    movel(p[x_c + 0.003071, y_c + 0.108854, z_c, rx, ry, rz], a, v)
    movel(p[x_c + 0.002863, y_c + 0.109126, z_c, rx, ry, rz], a, v)
    movel(p[x_c + 0.002653, y_c + 0.109393, z_c, rx, ry, rz], a, v)
    movel(p[x_c + 0.002442, y_c + 0.109655, z_c, rx, ry, rz], a, v)
    movel(p[x_c + 0.002230, y_c + 0.109912, z_c, rx, ry, rz], a, v)
    movel(p[x_c + 0.002017, y_c + 0.110165, z_c, rx, ry, rz], a, v)
    movel(p[x_c + 0.001803, y_c + 0.110413, z_c, rx, ry, rz], a, v)
    movel(p[x_c + 0.001589, y_c + 0.110656, z_c, rx, ry, rz], a, v)
    movel(p[x_c + 0.001373, y_c + 0.110893, z_c, rx, ry, rz], a, v)
    movel(p[x_c + 0.001157, y_c + 0.111126, z_c, rx, ry, rz], a, v)
    movel(p[x_c + 0.000939, y_c + 0.111354, z_c, rx, ry, rz], a, v)
    movel(p[x_c + 0.000722, y_c + 0.111576, z_c, rx, ry, rz], a, v)
    movel(p[x_c + 0.000503, y_c + 0.111793, z_c, rx, ry, rz], a, v)
    movel(p[x_c + 0.000284, y_c + 0.112005, z_c, rx, ry, rz], a, v)
    movel(p[x_c + 0.000064, y_c + 0.112211, z_c, rx, ry, rz], a, v)
    movel(p[x_c + -0.000156, y_c + 0.112412, z_c, rx, ry, rz], a, v)
    movel(p[x_c + -0.000377, y_c + 0.112608, z_c, rx, ry, rz], a, v)
    movel(p[x_c + -0.000598, y_c + 0.112798, z_c, rx, ry, rz], a, v)
    movel(p[x_c + -0.000820, y_c + 0.112982, z_c, rx, ry, rz], a, v)
    movel(p[x_c + -0.001042, y_c + 0.113161, z_c, rx, ry, rz], a, v)
    movel(p[x_c + -0.001264, y_c + 0.113334, z_c, rx, ry, rz], a, v)
    movel(p[x_c + -0.001487, y_c + 0.113501, z_c, rx, ry, rz], a, v)
    movel(p[x_c + -0.001709, y_c + 0.113662, z_c, rx, ry, rz], a, v)
    movel(p[x_c + -0.001932, y_c + 0.113818, z_c, rx, ry, rz], a, v)
    movel(p[x_c + -0.002155, y_c + 0.113967, z_c, rx, ry, rz], a, v)
    movel(p[x_c + -0.002378, y_c + 0.114111, z_c, rx, ry, rz], a, v)
    movel(p[x_c + -0.002600, y_c + 0.114248, z_c, rx, ry, rz], a, v)
    movel(p[x_c + -0.002823, y_c + 0.114380, z_c, rx, ry, rz], a, v)
    movel(p[x_c + -0.003046, y_c + 0.114505, z_c, rx, ry, rz], a, v)
    movel(p[x_c + -0.003268, y_c + 0.114624, z_c, rx, ry, rz], a, v)
    movel(p[x_c + -0.003491, y_c + 0.114737, z_c, rx, ry, rz], a, v)
    movel(p[x_c + -0.003491, y_c + 0.114737, z_c, rx, ry, rz], a, v)
    movel(p[x_c + -0.003766, y_c + 0.114868, z_c, rx, ry, rz], a, v)
    movel(p[x_c + -0.004040, y_c + 0.114986, z_c, rx, ry, rz], a, v)
    movel(p[x_c + -0.004311, y_c + 0.115094, z_c, rx, ry, rz], a, v)
    movel(p[x_c + -0.004579, y_c + 0.115189, z_c, rx, ry, rz], a, v)
    movel(p[x_c + -0.004844, y_c + 0.115274, z_c, rx, ry, rz], a, v)
    movel(p[x_c + -0.005105, y_c + 0.115347, z_c, rx, ry, rz], a, v)
    movel(p[x_c + -0.005364, y_c + 0.115408, z_c, rx, ry, rz], a, v)
    movel(p[x_c + -0.005619, y_c + 0.115459, z_c, rx, ry, rz], a, v)
    movel(p[x_c + -0.005870, y_c + 0.115499, z_c, rx, ry, rz], a, v)
    movel(p[x_c + -0.006117, y_c + 0.115529, z_c, rx, ry, rz], a, v)
    movel(p[x_c + -0.006360, y_c + 0.115547, z_c, rx, ry, rz], a, v)
    movel(p[x_c + -0.006599, y_c + 0.115556, z_c, rx, ry, rz], a, v)
    movel(p[x_c + -0.006833, y_c + 0.115553, z_c, rx, ry, rz], a, v)
    movel(p[x_c + -0.007062, y_c + 0.115541, z_c, rx, ry, rz], a, v)
    movel(p[x_c + -0.007287, y_c + 0.115519, z_c, rx, ry, rz], a, v)
    movel(p[x_c + -0.007506, y_c + 0.115486, z_c, rx, ry, rz], a, v)
    movel(p[x_c + -0.007720, y_c + 0.115444, z_c, rx, ry, rz], a, v)
    movel(p[x_c + -0.007929, y_c + 0.115393, z_c, rx, ry, rz], a, v)
    movel(p[x_c + -0.008132, y_c + 0.115331, z_c, rx, ry, rz], a, v)
    movel(p[x_c + -0.008329, y_c + 0.115261, z_c, rx, ry, rz], a, v)
    movel(p[x_c + -0.008521, y_c + 0.115181, z_c, rx, ry, rz], a, v)
    movel(p[x_c + -0.008705, y_c + 0.115092, z_c, rx, ry, rz], a, v)
    movel(p[x_c + -0.008884, y_c + 0.114994, z_c, rx, ry, rz], a, v)
    movel(p[x_c + -0.009056, y_c + 0.114887, z_c, rx, ry, rz], a, v)
    movel(p[x_c + -0.009221, y_c + 0.114771, z_c, rx, ry, rz], a, v)
    movel(p[x_c + -0.009379, y_c + 0.114647, z_c, rx, ry, rz], a, v)
    movel(p[x_c + -0.009530, y_c + 0.114514, z_c, rx, ry, rz], a, v)
    movel(p[x_c + -0.009674, y_c + 0.114373, z_c, rx, ry, rz], a, v)
    movel(p[x_c + -0.009809, y_c + 0.114224, z_c, rx, ry, rz], a, v)
    movel(p[x_c + -0.009938, y_c + 0.114066, z_c, rx, ry, rz], a, v)
    movel(p[x_c + -0.010058, y_c + 0.113901, z_c, rx, ry, rz], a, v)
    movel(p[x_c + -0.010170, y_c + 0.113728, z_c, rx, ry, rz], a, v)
    movel(p[x_c + -0.010274, y_c + 0.113547, z_c, rx, ry, rz], a, v)
    movel(p[x_c + -0.010369, y_c + 0.113359, z_c, rx, ry, rz], a, v)
    movel(p[x_c + -0.010456, y_c + 0.113164, z_c, rx, ry, rz], a, v)
    movel(p[x_c + -0.010533, y_c + 0.112961, z_c, rx, ry, rz], a, v)
    movel(p[x_c + -0.010602, y_c + 0.112751, z_c, rx, ry, rz], a, v)
    movel(p[x_c + -0.010661, y_c + 0.112534, z_c, rx, ry, rz], a, v)
    movel(p[x_c + -0.010711, y_c + 0.112310, z_c, rx, ry, rz], a, v)
    movel(p[x_c + -0.010751, y_c + 0.112079, z_c, rx, ry, rz], a, v)
    movel(p[x_c + -0.010782, y_c + 0.111842, z_c, rx, ry, rz], a, v)
    movel(p[x_c + -0.010802, y_c + 0.111598, z_c, rx, ry, rz], a, v)
    movel(p[x_c + -0.010812, y_c + 0.111349, z_c, rx, ry, rz], a, v)
    movel(p[x_c + -0.010812, y_c + 0.111092, z_c, rx, ry, rz], a, v)
    movel(p[x_c + -0.010801, y_c + 0.110830, z_c, rx, ry, rz], a, v)
    movel(p[x_c + -0.010779, y_c + 0.110562, z_c, rx, ry, rz], a, v)
    movel(p[x_c + -0.010746, y_c + 0.110288, z_c, rx, ry, rz], a, v)
    movel(p[x_c + -0.010702, y_c + 0.110008, z_c, rx, ry, rz], a, v)
    movel(p[x_c + -0.010647, y_c + 0.109723, z_c, rx, ry, rz], a, v)
    movel(p[x_c + -0.010647, y_c + 0.109723, z_c, rx, ry, rz], a, v)
    movel(p[x_c + -0.010635, y_c + 0.109670, z_c, rx, ry, rz], a, v)
    movel(p[x_c + -0.010621, y_c + 0.109614, z_c, rx, ry, rz], a, v)
    movel(p[x_c + -0.010606, y_c + 0.109555, z_c, rx, ry, rz], a, v)
    movel(p[x_c + -0.010588, y_c + 0.109492, z_c, rx, ry, rz], a, v)
    movel(p[x_c + -0.010569, y_c + 0.109426, z_c, rx, ry, rz], a, v)
    movel(p[x_c + -0.010548, y_c + 0.109356, z_c, rx, ry, rz], a, v)
    movel(p[x_c + -0.010525, y_c + 0.109284, z_c, rx, ry, rz], a, v)
    movel(p[x_c + -0.010501, y_c + 0.109209, z_c, rx, ry, rz], a, v)
    movel(p[x_c + -0.010475, y_c + 0.109130, z_c, rx, ry, rz], a, v)
    movel(p[x_c + -0.010447, y_c + 0.109049, z_c, rx, ry, rz], a, v)
    movel(p[x_c + -0.010417, y_c + 0.108965, z_c, rx, ry, rz], a, v)
    movel(p[x_c + -0.010386, y_c + 0.108878, z_c, rx, ry, rz], a, v)
    movel(p[x_c + -0.010353, y_c + 0.108788, z_c, rx, ry, rz], a, v)
    movel(p[x_c + -0.010318, y_c + 0.108695, z_c, rx, ry, rz], a, v)
    movel(p[x_c + -0.010282, y_c + 0.108600, z_c, rx, ry, rz], a, v)
    movel(p[x_c + -0.010244, y_c + 0.108502, z_c, rx, ry, rz], a, v)
    movel(p[x_c + -0.010205, y_c + 0.108401, z_c, rx, ry, rz], a, v)
    movel(p[x_c + -0.010164, y_c + 0.108298, z_c, rx, ry, rz], a, v)
    movel(p[x_c + -0.010122, y_c + 0.108192, z_c, rx, ry, rz], a, v)
    movel(p[x_c + -0.010078, y_c + 0.108084, z_c, rx, ry, rz], a, v)
    movel(p[x_c + -0.010033, y_c + 0.107973, z_c, rx, ry, rz], a, v)
    movel(p[x_c + -0.009986, y_c + 0.107860, z_c, rx, ry, rz], a, v)
    movel(p[x_c + -0.009938, y_c + 0.107745, z_c, rx, ry, rz], a, v)
    movel(p[x_c + -0.009888, y_c + 0.107627, z_c, rx, ry, rz], a, v)
    movel(p[x_c + -0.009837, y_c + 0.107507, z_c, rx, ry, rz], a, v)
    movel(p[x_c + -0.009784, y_c + 0.107385, z_c, rx, ry, rz], a, v)
    movel(p[x_c + -0.009731, y_c + 0.107261, z_c, rx, ry, rz], a, v)
    movel(p[x_c + -0.009676, y_c + 0.107135, z_c, rx, ry, rz], a, v)
    movel(p[x_c + -0.009619, y_c + 0.107007, z_c, rx, ry, rz], a, v)
    movel(p[x_c + -0.009561, y_c + 0.106877, z_c, rx, ry, rz], a, v)
    movel(p[x_c + -0.009503, y_c + 0.106744, z_c, rx, ry, rz], a, v)
    movel(p[x_c + -0.009442, y_c + 0.106610, z_c, rx, ry, rz], a, v)
    movel(p[x_c + -0.009381, y_c + 0.106475, z_c, rx, ry, rz], a, v)
    movel(p[x_c + -0.009318, y_c + 0.106337, z_c, rx, ry, rz], a, v)
    movel(p[x_c + -0.009254, y_c + 0.106198, z_c, rx, ry, rz], a, v)
    movel(p[x_c + -0.009189, y_c + 0.106057, z_c, rx, ry, rz], a, v)
    movel(p[x_c + -0.009123, y_c + 0.105914, z_c, rx, ry, rz], a, v)
    movel(p[x_c + -0.009056, y_c + 0.105770, z_c, rx, ry, rz], a, v)
    movel(p[x_c + -0.008988, y_c + 0.105624, z_c, rx, ry, rz], a, v)
    movel(p[x_c + -0.008918, y_c + 0.105476, z_c, rx, ry, rz], a, v)
    movel(p[x_c + -0.008848, y_c + 0.105328, z_c, rx, ry, rz], a, v)
    movel(p[x_c + -0.008776, y_c + 0.105178, z_c, rx, ry, rz], a, v)
    movel(p[x_c + -0.008704, y_c + 0.105026, z_c, rx, ry, rz], a, v)
    movel(p[x_c + -0.008630, y_c + 0.104873, z_c, rx, ry, rz], a, v)
    movel(p[x_c + -0.008555, y_c + 0.104719, z_c, rx, ry, rz], a, v)
    movel(p[x_c + -0.008480, y_c + 0.104564, z_c, rx, ry, rz], a, v)
    movel(p[x_c + -0.008403, y_c + 0.104408, z_c, rx, ry, rz], a, v)
    movel(p[x_c + -0.008326, y_c + 0.104251, z_c, rx, ry, rz], a, v)
    movel(p[x_c + -0.008248, y_c + 0.104092, z_c, rx, ry, rz], a, v)
    movel(p[x_c + -0.008248, y_c + 0.104092, z_c, rx, ry, rz], a, v)
    movel(p[x_c + -0.008098, y_c + 0.103789, z_c, rx, ry, rz], a, v)
    movel(p[x_c + -0.007954, y_c + 0.103496, z_c, rx, ry, rz], a, v)
    movel(p[x_c + -0.007814, y_c + 0.103212, z_c, rx, ry, rz], a, v)
    movel(p[x_c + -0.007679, y_c + 0.102937, z_c, rx, ry, rz], a, v)
    movel(p[x_c + -0.007549, y_c + 0.102670, z_c, rx, ry, rz], a, v)
    movel(p[x_c + -0.007424, y_c + 0.102412, z_c, rx, ry, rz], a, v)
    movel(p[x_c + -0.007303, y_c + 0.102162, z_c, rx, ry, rz], a, v)
    movel(p[x_c + -0.007187, y_c + 0.101920, z_c, rx, ry, rz], a, v)
    movel(p[x_c + -0.007075, y_c + 0.101686, z_c, rx, ry, rz], a, v)
    movel(p[x_c + -0.006968, y_c + 0.101459, z_c, rx, ry, rz], a, v)
    movel(p[x_c + -0.006864, y_c + 0.101239, z_c, rx, ry, rz], a, v)
    movel(p[x_c + -0.006765, y_c + 0.101026, z_c, rx, ry, rz], a, v)
    movel(p[x_c + -0.006670, y_c + 0.100820, z_c, rx, ry, rz], a, v)
    movel(p[x_c + -0.006578, y_c + 0.100620, z_c, rx, ry, rz], a, v)
    movel(p[x_c + -0.006491, y_c + 0.100427, z_c, rx, ry, rz], a, v)
    movel(p[x_c + -0.006407, y_c + 0.100240, z_c, rx, ry, rz], a, v)
    movel(p[x_c + -0.006327, y_c + 0.100058, z_c, rx, ry, rz], a, v)
    movel(p[x_c + -0.006251, y_c + 0.099882, z_c, rx, ry, rz], a, v)
    movel(p[x_c + -0.006178, y_c + 0.099711, z_c, rx, ry, rz], a, v)
    movel(p[x_c + -0.006108, y_c + 0.099545, z_c, rx, ry, rz], a, v)
    movel(p[x_c + -0.006042, y_c + 0.099384, z_c, rx, ry, rz], a, v)
    movel(p[x_c + -0.005979, y_c + 0.099227, z_c, rx, ry, rz], a, v)
    movel(p[x_c + -0.005919, y_c + 0.099075, z_c, rx, ry, rz], a, v)
    movel(p[x_c + -0.005862, y_c + 0.098926, z_c, rx, ry, rz], a, v)
    movel(p[x_c + -0.005808, y_c + 0.098782, z_c, rx, ry, rz], a, v)
    movel(p[x_c + -0.005756, y_c + 0.098641, z_c, rx, ry, rz], a, v)
    movel(p[x_c + -0.005708, y_c + 0.098503, z_c, rx, ry, rz], a, v)
    movel(p[x_c + -0.005662, y_c + 0.098368, z_c, rx, ry, rz], a, v)
    movel(p[x_c + -0.005619, y_c + 0.098236, z_c, rx, ry, rz], a, v)
    movel(p[x_c + -0.005578, y_c + 0.098107, z_c, rx, ry, rz], a, v)
    movel(p[x_c + -0.005540, y_c + 0.097980, z_c, rx, ry, rz], a, v)
    movel(p[x_c + -0.005504, y_c + 0.097855, z_c, rx, ry, rz], a, v)
    movel(p[x_c + -0.005470, y_c + 0.097732, z_c, rx, ry, rz], a, v)
    movel(p[x_c + -0.005438, y_c + 0.097610, z_c, rx, ry, rz], a, v)
    movel(p[x_c + -0.005408, y_c + 0.097490, z_c, rx, ry, rz], a, v)
    movel(p[x_c + -0.005381, y_c + 0.097371, z_c, rx, ry, rz], a, v)
    movel(p[x_c + -0.005355, y_c + 0.097253, z_c, rx, ry, rz], a, v)
    movel(p[x_c + -0.005331, y_c + 0.097136, z_c, rx, ry, rz], a, v)
    movel(p[x_c + -0.005308, y_c + 0.097018, z_c, rx, ry, rz], a, v)
    movel(p[x_c + -0.005287, y_c + 0.096901, z_c, rx, ry, rz], a, v)
    movel(p[x_c + -0.005268, y_c + 0.096784, z_c, rx, ry, rz], a, v)
    movel(p[x_c + -0.005250, y_c + 0.096667, z_c, rx, ry, rz], a, v)
    movel(p[x_c + -0.005233, y_c + 0.096549, z_c, rx, ry, rz], a, v)
    movel(p[x_c + -0.005217, y_c + 0.096430, z_c, rx, ry, rz], a, v)
    movel(p[x_c + -0.005203, y_c + 0.096310, z_c, rx, ry, rz], a, v)
    movel(p[x_c + -0.005189, y_c + 0.096188, z_c, rx, ry, rz], a, v)
    movel(p[x_c + -0.005177, y_c + 0.096065, z_c, rx, ry, rz], a, v)
    movel(p[x_c + -0.005165, y_c + 0.095941, z_c, rx, ry, rz], a, v)
    movel(p[x_c + -0.005154, y_c + 0.095814, z_c, rx, ry, rz], a, v)
    movel(p[x_c + -0.005154, y_c + 0.095814, z_c, rx, ry, rz], a, v)
    movel(p[x_c + -0.005139, y_c + 0.095611, z_c, rx, ry, rz], a, v)
    movel(p[x_c + -0.005127, y_c + 0.095410, z_c, rx, ry, rz], a, v)
    movel(p[x_c + -0.005119, y_c + 0.095210, z_c, rx, ry, rz], a, v)
    movel(p[x_c + -0.005114, y_c + 0.095010, z_c, rx, ry, rz], a, v)
    movel(p[x_c + -0.005113, y_c + 0.094812, z_c, rx, ry, rz], a, v)
    movel(p[x_c + -0.005115, y_c + 0.094615, z_c, rx, ry, rz], a, v)
    movel(p[x_c + -0.005120, y_c + 0.094419, z_c, rx, ry, rz], a, v)
    movel(p[x_c + -0.005129, y_c + 0.094224, z_c, rx, ry, rz], a, v)
    movel(p[x_c + -0.005141, y_c + 0.094030, z_c, rx, ry, rz], a, v)
    movel(p[x_c + -0.005156, y_c + 0.093837, z_c, rx, ry, rz], a, v)
    movel(p[x_c + -0.005175, y_c + 0.093646, z_c, rx, ry, rz], a, v)
    movel(p[x_c + -0.005197, y_c + 0.093455, z_c, rx, ry, rz], a, v)
    movel(p[x_c + -0.005223, y_c + 0.093266, z_c, rx, ry, rz], a, v)
    movel(p[x_c + -0.005252, y_c + 0.093077, z_c, rx, ry, rz], a, v)
    movel(p[x_c + -0.005284, y_c + 0.092890, z_c, rx, ry, rz], a, v)
    movel(p[x_c + -0.005320, y_c + 0.092704, z_c, rx, ry, rz], a, v)
    movel(p[x_c + -0.005359, y_c + 0.092519, z_c, rx, ry, rz], a, v)
    movel(p[x_c + -0.005401, y_c + 0.092335, z_c, rx, ry, rz], a, v)
    movel(p[x_c + -0.005447, y_c + 0.092153, z_c, rx, ry, rz], a, v)
    movel(p[x_c + -0.005496, y_c + 0.091971, z_c, rx, ry, rz], a, v)
    movel(p[x_c + -0.005548, y_c + 0.091791, z_c, rx, ry, rz], a, v)
    movel(p[x_c + -0.005604, y_c + 0.091612, z_c, rx, ry, rz], a, v)
    movel(p[x_c + -0.005663, y_c + 0.091434, z_c, rx, ry, rz], a, v)
    movel(p[x_c + -0.005726, y_c + 0.091257, z_c, rx, ry, rz], a, v)
    movel(p[x_c + -0.005792, y_c + 0.091082, z_c, rx, ry, rz], a, v)
    movel(p[x_c + -0.005861, y_c + 0.090907, z_c, rx, ry, rz], a, v)
    movel(p[x_c + -0.005934, y_c + 0.090734, z_c, rx, ry, rz], a, v)
    movel(p[x_c + -0.006010, y_c + 0.090562, z_c, rx, ry, rz], a, v)
    movel(p[x_c + -0.006089, y_c + 0.090392, z_c, rx, ry, rz], a, v)
    movel(p[x_c + -0.006171, y_c + 0.090222, z_c, rx, ry, rz], a, v)
    movel(p[x_c + -0.006257, y_c + 0.090054, z_c, rx, ry, rz], a, v)
    movel(p[x_c + -0.006347, y_c + 0.089887, z_c, rx, ry, rz], a, v)
    movel(p[x_c + -0.006439, y_c + 0.089721, z_c, rx, ry, rz], a, v)
    movel(p[x_c + -0.006535, y_c + 0.089556, z_c, rx, ry, rz], a, v)
    movel(p[x_c + -0.006634, y_c + 0.089393, z_c, rx, ry, rz], a, v)
    movel(p[x_c + -0.006737, y_c + 0.089231, z_c, rx, ry, rz], a, v)
    movel(p[x_c + -0.006843, y_c + 0.089070, z_c, rx, ry, rz], a, v)
    movel(p[x_c + -0.006952, y_c + 0.088911, z_c, rx, ry, rz], a, v)
    movel(p[x_c + -0.007064, y_c + 0.088752, z_c, rx, ry, rz], a, v)
    movel(p[x_c + -0.007180, y_c + 0.088595, z_c, rx, ry, rz], a, v)
    movel(p[x_c + -0.007299, y_c + 0.088440, z_c, rx, ry, rz], a, v)
    movel(p[x_c + -0.007422, y_c + 0.088285, z_c, rx, ry, rz], a, v)
    movel(p[x_c + -0.007547, y_c + 0.088132, z_c, rx, ry, rz], a, v)
    movel(p[x_c + -0.007677, y_c + 0.087980, z_c, rx, ry, rz], a, v)
    movel(p[x_c + -0.007809, y_c + 0.087830, z_c, rx, ry, rz], a, v)
    movel(p[x_c + -0.007945, y_c + 0.087681, z_c, rx, ry, rz], a, v)
    movel(p[x_c + -0.008083, y_c + 0.087533, z_c, rx, ry, rz], a, v)
    movel(p[x_c + -0.008226, y_c + 0.087386, z_c, rx, ry, rz], a, v)
    movel(p[x_c + -0.008371, y_c + 0.087241, z_c, rx, ry, rz], a, v)
    movel(p[x_c + -0.008371, y_c + 0.087241, z_c, rx, ry, rz], a, v)
    movel(p[x_c + -0.008488, y_c + 0.087127, z_c, rx, ry, rz], a, v)
    movel(p[x_c + -0.008605, y_c + 0.087016, z_c, rx, ry, rz], a, v)
    movel(p[x_c + -0.008723, y_c + 0.086906, z_c, rx, ry, rz], a, v)
    movel(p[x_c + -0.008842, y_c + 0.086798, z_c, rx, ry, rz], a, v)
    movel(p[x_c + -0.008961, y_c + 0.086692, z_c, rx, ry, rz], a, v)
    movel(p[x_c + -0.009082, y_c + 0.086587, z_c, rx, ry, rz], a, v)
    movel(p[x_c + -0.009203, y_c + 0.086484, z_c, rx, ry, rz], a, v)
    movel(p[x_c + -0.009326, y_c + 0.086383, z_c, rx, ry, rz], a, v)
    movel(p[x_c + -0.009450, y_c + 0.086283, z_c, rx, ry, rz], a, v)
    movel(p[x_c + -0.009576, y_c + 0.086184, z_c, rx, ry, rz], a, v)
    movel(p[x_c + -0.009704, y_c + 0.086087, z_c, rx, ry, rz], a, v)
    movel(p[x_c + -0.009833, y_c + 0.085990, z_c, rx, ry, rz], a, v)
    movel(p[x_c + -0.009964, y_c + 0.085895, z_c, rx, ry, rz], a, v)
    movel(p[x_c + -0.010098, y_c + 0.085801, z_c, rx, ry, rz], a, v)
    movel(p[x_c + -0.010233, y_c + 0.085708, z_c, rx, ry, rz], a, v)
    movel(p[x_c + -0.010371, y_c + 0.085616, z_c, rx, ry, rz], a, v)
    movel(p[x_c + -0.010512, y_c + 0.085525, z_c, rx, ry, rz], a, v)
    movel(p[x_c + -0.010655, y_c + 0.085435, z_c, rx, ry, rz], a, v)
    movel(p[x_c + -0.010800, y_c + 0.085345, z_c, rx, ry, rz], a, v)
    movel(p[x_c + -0.010949, y_c + 0.085256, z_c, rx, ry, rz], a, v)
    movel(p[x_c + -0.011101, y_c + 0.085168, z_c, rx, ry, rz], a, v)
    movel(p[x_c + -0.011256, y_c + 0.085080, z_c, rx, ry, rz], a, v)
    movel(p[x_c + -0.011414, y_c + 0.084993, z_c, rx, ry, rz], a, v)
    movel(p[x_c + -0.011575, y_c + 0.084905, z_c, rx, ry, rz], a, v)
    movel(p[x_c + -0.011740, y_c + 0.084819, z_c, rx, ry, rz], a, v)
    movel(p[x_c + -0.011909, y_c + 0.084732, z_c, rx, ry, rz], a, v)
    movel(p[x_c + -0.012082, y_c + 0.084646, z_c, rx, ry, rz], a, v)
    movel(p[x_c + -0.012258, y_c + 0.084560, z_c, rx, ry, rz], a, v)
    movel(p[x_c + -0.012439, y_c + 0.084473, z_c, rx, ry, rz], a, v)
    movel(p[x_c + -0.012624, y_c + 0.084387, z_c, rx, ry, rz], a, v)
    movel(p[x_c + -0.012813, y_c + 0.084301, z_c, rx, ry, rz], a, v)
    movel(p[x_c + -0.013007, y_c + 0.084214, z_c, rx, ry, rz], a, v)
    movel(p[x_c + -0.013205, y_c + 0.084127, z_c, rx, ry, rz], a, v)
    movel(p[x_c + -0.013408, y_c + 0.084040, z_c, rx, ry, rz], a, v)
    movel(p[x_c + -0.013616, y_c + 0.083953, z_c, rx, ry, rz], a, v)
    movel(p[x_c + -0.013829, y_c + 0.083865, z_c, rx, ry, rz], a, v)
    movel(p[x_c + -0.014047, y_c + 0.083776, z_c, rx, ry, rz], a, v)
    movel(p[x_c + -0.014270, y_c + 0.083687, z_c, rx, ry, rz], a, v)
    movel(p[x_c + -0.014499, y_c + 0.083597, z_c, rx, ry, rz], a, v)
    movel(p[x_c + -0.014733, y_c + 0.083507, z_c, rx, ry, rz], a, v)
    movel(p[x_c + -0.014973, y_c + 0.083416, z_c, rx, ry, rz], a, v)
    movel(p[x_c + -0.015219, y_c + 0.083323, z_c, rx, ry, rz], a, v)
    movel(p[x_c + -0.015471, y_c + 0.083230, z_c, rx, ry, rz], a, v)
    movel(p[x_c + -0.015729, y_c + 0.083136, z_c, rx, ry, rz], a, v)
    movel(p[x_c + -0.015993, y_c + 0.083041, z_c, rx, ry, rz], a, v)
    movel(p[x_c + -0.016263, y_c + 0.082944, z_c, rx, ry, rz], a, v)
    movel(p[x_c + -0.016540, y_c + 0.082846, z_c, rx, ry, rz], a, v)
    movel(p[x_c + -0.016824, y_c + 0.082747, z_c, rx, ry, rz], a, v)
    movel(p[x_c + -0.017114, y_c + 0.082647, z_c, rx, ry, rz], a, v)
    movel(p[x_c + -0.017114, y_c + 0.082647, z_c, rx, ry, rz], a, v)
    movel(p[x_c + -0.017237, y_c + 0.082604, z_c, rx, ry, rz], a, v)
    movel(p[x_c + -0.017361, y_c + 0.082562, z_c, rx, ry, rz], a, v)
    movel(p[x_c + -0.017484, y_c + 0.082519, z_c, rx, ry, rz], a, v)
    movel(p[x_c + -0.017607, y_c + 0.082476, z_c, rx, ry, rz], a, v)
    movel(p[x_c + -0.017729, y_c + 0.082433, z_c, rx, ry, rz], a, v)
    movel(p[x_c + -0.017852, y_c + 0.082390, z_c, rx, ry, rz], a, v)
    movel(p[x_c + -0.017973, y_c + 0.082347, z_c, rx, ry, rz], a, v)
    movel(p[x_c + -0.018094, y_c + 0.082305, z_c, rx, ry, rz], a, v)
    movel(p[x_c + -0.018215, y_c + 0.082262, z_c, rx, ry, rz], a, v)
    movel(p[x_c + -0.018335, y_c + 0.082219, z_c, rx, ry, rz], a, v)
    movel(p[x_c + -0.018454, y_c + 0.082177, z_c, rx, ry, rz], a, v)
    movel(p[x_c + -0.018572, y_c + 0.082134, z_c, rx, ry, rz], a, v)
    movel(p[x_c + -0.018689, y_c + 0.082092, z_c, rx, ry, rz], a, v)
    movel(p[x_c + -0.018805, y_c + 0.082051, z_c, rx, ry, rz], a, v)
    movel(p[x_c + -0.018919, y_c + 0.082009, z_c, rx, ry, rz], a, v)
    movel(p[x_c + -0.019033, y_c + 0.081968, z_c, rx, ry, rz], a, v)
    movel(p[x_c + -0.019145, y_c + 0.081927, z_c, rx, ry, rz], a, v)
    movel(p[x_c + -0.019256, y_c + 0.081886, z_c, rx, ry, rz], a, v)
    movel(p[x_c + -0.019366, y_c + 0.081846, z_c, rx, ry, rz], a, v)
    movel(p[x_c + -0.019474, y_c + 0.081806, z_c, rx, ry, rz], a, v)
    movel(p[x_c + -0.019580, y_c + 0.081767, z_c, rx, ry, rz], a, v)
    movel(p[x_c + -0.019685, y_c + 0.081728, z_c, rx, ry, rz], a, v)
    movel(p[x_c + -0.019788, y_c + 0.081690, z_c, rx, ry, rz], a, v)
    movel(p[x_c + -0.019889, y_c + 0.081652, z_c, rx, ry, rz], a, v)
    movel(p[x_c + -0.019988, y_c + 0.081615, z_c, rx, ry, rz], a, v)
    movel(p[x_c + -0.020085, y_c + 0.081578, z_c, rx, ry, rz], a, v)
    movel(p[x_c + -0.020180, y_c + 0.081542, z_c, rx, ry, rz], a, v)
    movel(p[x_c + -0.020273, y_c + 0.081506, z_c, rx, ry, rz], a, v)
    movel(p[x_c + -0.020363, y_c + 0.081472, z_c, rx, ry, rz], a, v)
    movel(p[x_c + -0.020451, y_c + 0.081438, z_c, rx, ry, rz], a, v)
    movel(p[x_c + -0.020537, y_c + 0.081405, z_c, rx, ry, rz], a, v)
    movel(p[x_c + -0.020620, y_c + 0.081372, z_c, rx, ry, rz], a, v)
    movel(p[x_c + -0.020701, y_c + 0.081340, z_c, rx, ry, rz], a, v)
    movel(p[x_c + -0.020779, y_c + 0.081310, z_c, rx, ry, rz], a, v)
    movel(p[x_c + -0.020855, y_c + 0.081280, z_c, rx, ry, rz], a, v)
    movel(p[x_c + -0.020927, y_c + 0.081251, z_c, rx, ry, rz], a, v)
    movel(p[x_c + -0.020997, y_c + 0.081223, z_c, rx, ry, rz], a, v)
    movel(p[x_c + -0.021064, y_c + 0.081195, z_c, rx, ry, rz], a, v)
    movel(p[x_c + -0.021127, y_c + 0.081169, z_c, rx, ry, rz], a, v)
    movel(p[x_c + -0.021188, y_c + 0.081144, z_c, rx, ry, rz], a, v)
    movel(p[x_c + -0.021245, y_c + 0.081120, z_c, rx, ry, rz], a, v)
    movel(p[x_c + -0.021299, y_c + 0.081097, z_c, rx, ry, rz], a, v)
    movel(p[x_c + -0.021350, y_c + 0.081075, z_c, rx, ry, rz], a, v)
    movel(p[x_c + -0.021397, y_c + 0.081054, z_c, rx, ry, rz], a, v)
    movel(p[x_c + -0.021441, y_c + 0.081034, z_c, rx, ry, rz], a, v)
    movel(p[x_c + -0.021481, y_c + 0.081016, z_c, rx, ry, rz], a, v)
    movel(p[x_c + -0.021517, y_c + 0.080999, z_c, rx, ry, rz], a, v)
    movel(p[x_c + -0.021550, y_c + 0.080983, z_c, rx, ry, rz], a, v)
    movel(p[x_c + -0.021579, y_c + 0.080968, z_c, rx, ry, rz], a, v)
    movel(p[x_c + -0.021579, y_c + 0.080968, z_c, rx, ry, rz], a, v)
    movel(p[x_c + -0.022375, y_c + 0.080552, z_c, rx, ry, rz], a, v)
    movel(p[x_c + -0.022375, y_c + 0.080552, z_c, rx, ry, rz], a, v)
    movel(p[x_c + -0.020813, y_c + 0.080676, z_c, rx, ry, rz], a, v)
    movel(p[x_c + -0.020813, y_c + 0.080676, z_c, rx, ry, rz], a, v)
    movel(p[x_c + -0.020726, y_c + 0.080682, z_c, rx, ry, rz], a, v)
    movel(p[x_c + -0.020631, y_c + 0.080688, z_c, rx, ry, rz], a, v)
    movel(p[x_c + -0.020530, y_c + 0.080692, z_c, rx, ry, rz], a, v)
    movel(p[x_c + -0.020422, y_c + 0.080697, z_c, rx, ry, rz], a, v)
    movel(p[x_c + -0.020307, y_c + 0.080700, z_c, rx, ry, rz], a, v)
    movel(p[x_c + -0.020184, y_c + 0.080703, z_c, rx, ry, rz], a, v)
    movel(p[x_c + -0.020055, y_c + 0.080704, z_c, rx, ry, rz], a, v)
    movel(p[x_c + -0.019919, y_c + 0.080706, z_c, rx, ry, rz], a, v)
    movel(p[x_c + -0.019775, y_c + 0.080706, z_c, rx, ry, rz], a, v)
    movel(p[x_c + -0.019625, y_c + 0.080706, z_c, rx, ry, rz], a, v)
    movel(p[x_c + -0.019466, y_c + 0.080705, z_c, rx, ry, rz], a, v)
    movel(p[x_c + -0.019301, y_c + 0.080703, z_c, rx, ry, rz], a, v)
    movel(p[x_c + -0.019128, y_c + 0.080700, z_c, rx, ry, rz], a, v)
    movel(p[x_c + -0.018948, y_c + 0.080697, z_c, rx, ry, rz], a, v)
    movel(p[x_c + -0.018760, y_c + 0.080692, z_c, rx, ry, rz], a, v)
    movel(p[x_c + -0.018565, y_c + 0.080688, z_c, rx, ry, rz], a, v)
    movel(p[x_c + -0.018362, y_c + 0.080682, z_c, rx, ry, rz], a, v)
    movel(p[x_c + -0.018152, y_c + 0.080675, z_c, rx, ry, rz], a, v)
    movel(p[x_c + -0.017933, y_c + 0.080668, z_c, rx, ry, rz], a, v)
    movel(p[x_c + -0.017707, y_c + 0.080660, z_c, rx, ry, rz], a, v)
    movel(p[x_c + -0.017474, y_c + 0.080651, z_c, rx, ry, rz], a, v)
    movel(p[x_c + -0.017232, y_c + 0.080642, z_c, rx, ry, rz], a, v)
    movel(p[x_c + -0.016982, y_c + 0.080632, z_c, rx, ry, rz], a, v)
    movel(p[x_c + -0.016724, y_c + 0.080620, z_c, rx, ry, rz], a, v)
    movel(p[x_c + -0.016459, y_c + 0.080609, z_c, rx, ry, rz], a, v)
    movel(p[x_c + -0.016185, y_c + 0.080596, z_c, rx, ry, rz], a, v)
    movel(p[x_c + -0.015903, y_c + 0.080582, z_c, rx, ry, rz], a, v)
    movel(p[x_c + -0.015613, y_c + 0.080568, z_c, rx, ry, rz], a, v)
    movel(p[x_c + -0.015314, y_c + 0.080553, z_c, rx, ry, rz], a, v)
    movel(p[x_c + -0.015008, y_c + 0.080537, z_c, rx, ry, rz], a, v)
    movel(p[x_c + -0.014693, y_c + 0.080520, z_c, rx, ry, rz], a, v)
    movel(p[x_c + -0.014369, y_c + 0.080503, z_c, rx, ry, rz], a, v)
    movel(p[x_c + -0.014037, y_c + 0.080485, z_c, rx, ry, rz], a, v)
    movel(p[x_c + -0.013697, y_c + 0.080466, z_c, rx, ry, rz], a, v)
    movel(p[x_c + -0.013348, y_c + 0.080446, z_c, rx, ry, rz], a, v)
    movel(p[x_c + -0.012990, y_c + 0.080425, z_c, rx, ry, rz], a, v)
    movel(p[x_c + -0.012624, y_c + 0.080403, z_c, rx, ry, rz], a, v)
    movel(p[x_c + -0.012249, y_c + 0.080381, z_c, rx, ry, rz], a, v)
    movel(p[x_c + -0.011865, y_c + 0.080358, z_c, rx, ry, rz], a, v)
    movel(p[x_c + -0.011472, y_c + 0.080334, z_c, rx, ry, rz], a, v)
    movel(p[x_c + -0.011070, y_c + 0.080309, z_c, rx, ry, rz], a, v)
    movel(p[x_c + -0.010660, y_c + 0.080283, z_c, rx, ry, rz], a, v)
    movel(p[x_c + -0.010240, y_c + 0.080257, z_c, rx, ry, rz], a, v)
    movel(p[x_c + -0.009811, y_c + 0.080230, z_c, rx, ry, rz], a, v)
    movel(p[x_c + -0.009374, y_c + 0.080201, z_c, rx, ry, rz], a, v)
    movel(p[x_c + -0.008927, y_c + 0.080172, z_c, rx, ry, rz], a, v)
    movel(p[x_c + -0.008471, y_c + 0.080143, z_c, rx, ry, rz], a, v)
    movel(p[x_c + -0.008005, y_c + 0.080112, z_c, rx, ry, rz], a, v)
    movel(p[x_c + -0.007530, y_c + 0.080080, z_c, rx, ry, rz], a, v)
    movel(p[x_c + -0.007530, y_c + 0.080080, z_c, rx, ry, rz], a, v)
    movel(p[x_c + -0.007298, y_c + 0.080065, z_c, rx, ry, rz], a, v)
    movel(p[x_c + -0.007064, y_c + 0.080051, z_c, rx, ry, rz], a, v)
    movel(p[x_c + -0.006828, y_c + 0.080037, z_c, rx, ry, rz], a, v)
    movel(p[x_c + -0.006591, y_c + 0.080024, z_c, rx, ry, rz], a, v)
    movel(p[x_c + -0.006353, y_c + 0.080011, z_c, rx, ry, rz], a, v)
    movel(p[x_c + -0.006115, y_c + 0.079999, z_c, rx, ry, rz], a, v)
    movel(p[x_c + -0.005875, y_c + 0.079988, z_c, rx, ry, rz], a, v)
    movel(p[x_c + -0.005635, y_c + 0.079977, z_c, rx, ry, rz], a, v)
    movel(p[x_c + -0.005395, y_c + 0.079967, z_c, rx, ry, rz], a, v)
    movel(p[x_c + -0.005155, y_c + 0.079958, z_c, rx, ry, rz], a, v)
    movel(p[x_c + -0.004915, y_c + 0.079949, z_c, rx, ry, rz], a, v)
    movel(p[x_c + -0.004675, y_c + 0.079941, z_c, rx, ry, rz], a, v)
    movel(p[x_c + -0.004436, y_c + 0.079934, z_c, rx, ry, rz], a, v)
    movel(p[x_c + -0.004198, y_c + 0.079927, z_c, rx, ry, rz], a, v)
    movel(p[x_c + -0.003960, y_c + 0.079921, z_c, rx, ry, rz], a, v)
    movel(p[x_c + -0.003724, y_c + 0.079916, z_c, rx, ry, rz], a, v)
    movel(p[x_c + -0.003489, y_c + 0.079911, z_c, rx, ry, rz], a, v)
    movel(p[x_c + -0.003255, y_c + 0.079907, z_c, rx, ry, rz], a, v)
    movel(p[x_c + -0.003023, y_c + 0.079903, z_c, rx, ry, rz], a, v)
    movel(p[x_c + -0.002793, y_c + 0.079900, z_c, rx, ry, rz], a, v)
    movel(p[x_c + -0.002565, y_c + 0.079898, z_c, rx, ry, rz], a, v)
    movel(p[x_c + -0.002339, y_c + 0.079896, z_c, rx, ry, rz], a, v)
    movel(p[x_c + -0.002116, y_c + 0.079895, z_c, rx, ry, rz], a, v)
    movel(p[x_c + -0.001895, y_c + 0.079895, z_c, rx, ry, rz], a, v)
    movel(p[x_c + -0.001678, y_c + 0.079895, z_c, rx, ry, rz], a, v)
    movel(p[x_c + -0.001463, y_c + 0.079896, z_c, rx, ry, rz], a, v)
    movel(p[x_c + -0.001252, y_c + 0.079898, z_c, rx, ry, rz], a, v)
    movel(p[x_c + -0.001044, y_c + 0.079900, z_c, rx, ry, rz], a, v)
    movel(p[x_c + -0.000840, y_c + 0.079903, z_c, rx, ry, rz], a, v)
    movel(p[x_c + -0.000640, y_c + 0.079906, z_c, rx, ry, rz], a, v)
    movel(p[x_c + -0.000443, y_c + 0.079910, z_c, rx, ry, rz], a, v)
    movel(p[x_c + -0.000251, y_c + 0.079915, z_c, rx, ry, rz], a, v)
    movel(p[x_c + -0.000064, y_c + 0.079920, z_c, rx, ry, rz], a, v)
    movel(p[x_c + 0.000119, y_c + 0.079926, z_c, rx, ry, rz], a, v)
    movel(p[x_c + 0.000297, y_c + 0.079933, z_c, rx, ry, rz], a, v)
    movel(p[x_c + 0.000470, y_c + 0.079940, z_c, rx, ry, rz], a, v)
    movel(p[x_c + 0.000638, y_c + 0.079948, z_c, rx, ry, rz], a, v)
    movel(p[x_c + 0.000800, y_c + 0.079957, z_c, rx, ry, rz], a, v)
    movel(p[x_c + 0.000957, y_c + 0.079966, z_c, rx, ry, rz], a, v)
    movel(p[x_c + 0.001108, y_c + 0.079976, z_c, rx, ry, rz], a, v)
    movel(p[x_c + 0.001253, y_c + 0.079986, z_c, rx, ry, rz], a, v)
    movel(p[x_c + 0.001392, y_c + 0.079998, z_c, rx, ry, rz], a, v)
    movel(p[x_c + 0.001524, y_c + 0.080009, z_c, rx, ry, rz], a, v)
    movel(p[x_c + 0.001650, y_c + 0.080022, z_c, rx, ry, rz], a, v)
    movel(p[x_c + 0.001769, y_c + 0.080035, z_c, rx, ry, rz], a, v)
    movel(p[x_c + 0.001881, y_c + 0.080048, z_c, rx, ry, rz], a, v)
    movel(p[x_c + 0.001985, y_c + 0.080063, z_c, rx, ry, rz], a, v)
    movel(p[x_c + 0.002083, y_c + 0.080077, z_c, rx, ry, rz], a, v)
    movel(p[x_c + 0.002172, y_c + 0.080093, z_c, rx, ry, rz], a, v)
    movel(p[x_c + 0.002172, y_c + 0.080093, z_c, rx, ry, rz], a, v)
    movel(p[x_c + 0.002172, y_c + 0.080093, z_c, rx, ry, rz], a, v)
    movel(p[x_c + 0.002172, y_c + 0.080093, z_c, rx, ry, rz], a, v)
    movel(p[x_c + 0.002172, y_c + 0.080093, z_c, rx, ry, rz], a, v)
    movel(p[x_c + 0.002172, y_c + 0.080093, z_c, rx, ry, rz], a, v)
    movel(p[x_c + 0.002172, y_c + 0.080093, z_c, rx, ry, rz], a, v)
    movel(p[x_c + 0.002172, y_c + 0.080093, z_c, rx, ry, rz], a, v)
    movel(p[x_c + 0.002172, y_c + 0.080093, z_c, rx, ry, rz], a, v)
    movel(p[x_c + 0.002172, y_c + 0.080094, z_c, rx, ry, rz], a, v)
    movel(p[x_c + 0.002172, y_c + 0.080094, z_c, rx, ry, rz], a, v)
    movel(p[x_c + -0.072957, y_c + 0.089770, z_c, rx, ry, rz], a, v)
    movel(p[x_c + -0.072957, y_c + 0.089770, z_c, rx, ry, rz], a, v)
    movel(p[x_c + -0.072957, y_c + 0.089770, z_c, rx, ry, rz], a, v)
    movel(p[x_c + -0.072957, y_c + 0.089770, z_c, rx, ry, rz], a, v)
    movel(p[x_c + -0.072957, y_c + 0.089770, z_c, rx, ry, rz], a, v)
    movel(p[x_c + -0.072957, y_c + 0.089770, z_c, rx, ry, rz], a, v)
    movel(p[x_c + -0.072957, y_c + 0.089770, z_c, rx, ry, rz], a, v)
    movel(p[x_c + -0.072957, y_c + 0.089770, z_c, rx, ry, rz], a, v)
    movel(p[x_c + -0.072957, y_c + 0.089770, z_c, rx, ry, rz], a, v)
    movel(p[x_c + -0.072957, y_c + 0.089770, z_c, rx, ry, rz], a, v)
    movel(p[x_c + -0.072957, y_c + 0.089770, z_c, rx, ry, rz], a, v)
    movel(p[x_c + -0.072450, y_c + 0.089935, z_c, rx, ry, rz], a, v)
    movel(p[x_c + -0.071947, y_c + 0.090098, z_c, rx, ry, rz], a, v)
    movel(p[x_c + -0.071450, y_c + 0.090258, z_c, rx, ry, rz], a, v)
    movel(p[x_c + -0.070956, y_c + 0.090416, z_c, rx, ry, rz], a, v)
    movel(p[x_c + -0.070468, y_c + 0.090571, z_c, rx, ry, rz], a, v)
    movel(p[x_c + -0.069984, y_c + 0.090724, z_c, rx, ry, rz], a, v)
    movel(p[x_c + -0.069504, y_c + 0.090874, z_c, rx, ry, rz], a, v)
    movel(p[x_c + -0.069030, y_c + 0.091021, z_c, rx, ry, rz], a, v)
    movel(p[x_c + -0.068559, y_c + 0.091166, z_c, rx, ry, rz], a, v)
    movel(p[x_c + -0.068094, y_c + 0.091308, z_c, rx, ry, rz], a, v)
    movel(p[x_c + -0.067633, y_c + 0.091448, z_c, rx, ry, rz], a, v)
    movel(p[x_c + -0.067176, y_c + 0.091586, z_c, rx, ry, rz], a, v)
    movel(p[x_c + -0.066724, y_c + 0.091720, z_c, rx, ry, rz], a, v)
    movel(p[x_c + -0.066277, y_c + 0.091853, z_c, rx, ry, rz], a, v)
    movel(p[x_c + -0.065833, y_c + 0.091982, z_c, rx, ry, rz], a, v)
    movel(p[x_c + -0.065395, y_c + 0.092110, z_c, rx, ry, rz], a, v)
    movel(p[x_c + -0.064961, y_c + 0.092234, z_c, rx, ry, rz], a, v)
    movel(p[x_c + -0.064531, y_c + 0.092356, z_c, rx, ry, rz], a, v)
    movel(p[x_c + -0.064105, y_c + 0.092476, z_c, rx, ry, rz], a, v)
    movel(p[x_c + -0.063684, y_c + 0.092593, z_c, rx, ry, rz], a, v)
    movel(p[x_c + -0.063268, y_c + 0.092708, z_c, rx, ry, rz], a, v)
    movel(p[x_c + -0.062855, y_c + 0.092820, z_c, rx, ry, rz], a, v)
    movel(p[x_c + -0.062447, y_c + 0.092930, z_c, rx, ry, rz], a, v)
    movel(p[x_c + -0.062044, y_c + 0.093037, z_c, rx, ry, rz], a, v)
    movel(p[x_c + -0.061644, y_c + 0.093142, z_c, rx, ry, rz], a, v)
    movel(p[x_c + -0.061249, y_c + 0.093244, z_c, rx, ry, rz], a, v)
    movel(p[x_c + -0.060858, y_c + 0.093344, z_c, rx, ry, rz], a, v)
    movel(p[x_c + -0.060471, y_c + 0.093442, z_c, rx, ry, rz], a, v)
    movel(p[x_c + -0.060089, y_c + 0.093537, z_c, rx, ry, rz], a, v)
    movel(p[x_c + -0.059711, y_c + 0.093629, z_c, rx, ry, rz], a, v)
    movel(p[x_c + -0.059336, y_c + 0.093719, z_c, rx, ry, rz], a, v)
    movel(p[x_c + -0.058966, y_c + 0.093807, z_c, rx, ry, rz], a, v)
    movel(p[x_c + -0.058601, y_c + 0.093892, z_c, rx, ry, rz], a, v)
    movel(p[x_c + -0.058239, y_c + 0.093975, z_c, rx, ry, rz], a, v)
    movel(p[x_c + -0.057881, y_c + 0.094055, z_c, rx, ry, rz], a, v)
    movel(p[x_c + -0.057528, y_c + 0.094133, z_c, rx, ry, rz], a, v)
    movel(p[x_c + -0.057178, y_c + 0.094209, z_c, rx, ry, rz], a, v)
    movel(p[x_c + -0.056833, y_c + 0.094282, z_c, rx, ry, rz], a, v)
    movel(p[x_c + -0.056491, y_c + 0.094353, z_c, rx, ry, rz], a, v)
    movel(p[x_c + -0.056154, y_c + 0.094421, z_c, rx, ry, rz], a, v)
    movel(p[x_c + -0.055820, y_c + 0.094487, z_c, rx, ry, rz], a, v)
    movel(p[x_c + -0.055491, y_c + 0.094550, z_c, rx, ry, rz], a, v)
    movel(p[x_c + -0.055165, y_c + 0.094611, z_c, rx, ry, rz], a, v)
    movel(p[x_c + -0.054843, y_c + 0.094670, z_c, rx, ry, rz], a, v)
    movel(p[x_c + -0.054526, y_c + 0.094727, z_c, rx, ry, rz], a, v)
    movel(p[x_c + -0.054212, y_c + 0.094781, z_c, rx, ry, rz], a, v)
    movel(p[x_c + -0.053902, y_c + 0.094832, z_c, rx, ry, rz], a, v)
    movel(p[x_c + -0.053596, y_c + 0.094882, z_c, rx, ry, rz], a, v)
    movel(p[x_c + -0.053294, y_c + 0.094929, z_c, rx, ry, rz], a, v)
    movel(p[x_c + -0.053294, y_c + 0.094929, z_c, rx, ry, rz], a, v)
    movel(p[x_c + -0.053125, y_c + 0.094954, z_c, rx, ry, rz], a, v)
    movel(p[x_c + -0.052952, y_c + 0.094978, z_c, rx, ry, rz], a, v)
    movel(p[x_c + -0.052774, y_c + 0.095001, z_c, rx, ry, rz], a, v)
    movel(p[x_c + -0.052592, y_c + 0.095023, z_c, rx, ry, rz], a, v)
    movel(p[x_c + -0.052406, y_c + 0.095045, z_c, rx, ry, rz], a, v)
    movel(p[x_c + -0.052216, y_c + 0.095065, z_c, rx, ry, rz], a, v)
    movel(p[x_c + -0.052022, y_c + 0.095085, z_c, rx, ry, rz], a, v)
    movel(p[x_c + -0.051825, y_c + 0.095104, z_c, rx, ry, rz], a, v)
    movel(p[x_c + -0.051626, y_c + 0.095122, z_c, rx, ry, rz], a, v)
    movel(p[x_c + -0.051424, y_c + 0.095139, z_c, rx, ry, rz], a, v)
    movel(p[x_c + -0.051219, y_c + 0.095155, z_c, rx, ry, rz], a, v)
    movel(p[x_c + -0.051012, y_c + 0.095170, z_c, rx, ry, rz], a, v)
    movel(p[x_c + -0.050804, y_c + 0.095185, z_c, rx, ry, rz], a, v)
    movel(p[x_c + -0.050593, y_c + 0.095198, z_c, rx, ry, rz], a, v)
    movel(p[x_c + -0.050382, y_c + 0.095211, z_c, rx, ry, rz], a, v)
    movel(p[x_c + -0.050169, y_c + 0.095223, z_c, rx, ry, rz], a, v)
    movel(p[x_c + -0.049956, y_c + 0.095234, z_c, rx, ry, rz], a, v)
    movel(p[x_c + -0.049742, y_c + 0.095244, z_c, rx, ry, rz], a, v)
    movel(p[x_c + -0.049528, y_c + 0.095252, z_c, rx, ry, rz], a, v)
    movel(p[x_c + -0.049315, y_c + 0.095261, z_c, rx, ry, rz], a, v)
    movel(p[x_c + -0.049101, y_c + 0.095268, z_c, rx, ry, rz], a, v)
    movel(p[x_c + -0.048888, y_c + 0.095274, z_c, rx, ry, rz], a, v)
    movel(p[x_c + -0.048676, y_c + 0.095279, z_c, rx, ry, rz], a, v)
    movel(p[x_c + -0.048465, y_c + 0.095283, z_c, rx, ry, rz], a, v)
    movel(p[x_c + -0.048256, y_c + 0.095287, z_c, rx, ry, rz], a, v)
    movel(p[x_c + -0.048048, y_c + 0.095289, z_c, rx, ry, rz], a, v)
    movel(p[x_c + -0.047842, y_c + 0.095291, z_c, rx, ry, rz], a, v)
    movel(p[x_c + -0.047639, y_c + 0.095291, z_c, rx, ry, rz], a, v)
    movel(p[x_c + -0.047438, y_c + 0.095291, z_c, rx, ry, rz], a, v)
    movel(p[x_c + -0.047240, y_c + 0.095289, z_c, rx, ry, rz], a, v)
    movel(p[x_c + -0.047044, y_c + 0.095287, z_c, rx, ry, rz], a, v)
    movel(p[x_c + -0.046853, y_c + 0.095284, z_c, rx, ry, rz], a, v)
    movel(p[x_c + -0.046665, y_c + 0.095279, z_c, rx, ry, rz], a, v)
    movel(p[x_c + -0.046480, y_c + 0.095274, z_c, rx, ry, rz], a, v)
    movel(p[x_c + -0.046300, y_c + 0.095268, z_c, rx, ry, rz], a, v)
    movel(p[x_c + -0.046125, y_c + 0.095260, z_c, rx, ry, rz], a, v)
    movel(p[x_c + -0.045954, y_c + 0.095252, z_c, rx, ry, rz], a, v)
    movel(p[x_c + -0.045788, y_c + 0.095243, z_c, rx, ry, rz], a, v)
    movel(p[x_c + -0.045627, y_c + 0.095232, z_c, rx, ry, rz], a, v)
    movel(p[x_c + -0.045472, y_c + 0.095221, z_c, rx, ry, rz], a, v)
    movel(p[x_c + -0.045323, y_c + 0.095208, z_c, rx, ry, rz], a, v)
    movel(p[x_c + -0.045179, y_c + 0.095195, z_c, rx, ry, rz], a, v)
    movel(p[x_c + -0.045043, y_c + 0.095181, z_c, rx, ry, rz], a, v)
    movel(p[x_c + -0.044912, y_c + 0.095165, z_c, rx, ry, rz], a, v)
    movel(p[x_c + -0.044789, y_c + 0.095149, z_c, rx, ry, rz], a, v)
    movel(p[x_c + -0.044673, y_c + 0.095131, z_c, rx, ry, rz], a, v)
    movel(p[x_c + -0.044564, y_c + 0.095113, z_c, rx, ry, rz], a, v)
    movel(p[x_c + -0.044463, y_c + 0.095093, z_c, rx, ry, rz], a, v)
    movel(p[x_c + -0.044370, y_c + 0.095072, z_c, rx, ry, rz], a, v)
    movel(p[x_c + -0.044370, y_c + 0.095072, z_c, rx, ry, rz], a, v)
    movel(p[x_c + -0.044336, y_c + 0.095064, z_c, rx, ry, rz], a, v)
    movel(p[x_c + -0.044303, y_c + 0.095057, z_c, rx, ry, rz], a, v)
    movel(p[x_c + -0.044270, y_c + 0.095049, z_c, rx, ry, rz], a, v)
    movel(p[x_c + -0.044237, y_c + 0.095042, z_c, rx, ry, rz], a, v)
    movel(p[x_c + -0.044204, y_c + 0.095035, z_c, rx, ry, rz], a, v)
    movel(p[x_c + -0.044171, y_c + 0.095028, z_c, rx, ry, rz], a, v)
    movel(p[x_c + -0.044139, y_c + 0.095021, z_c, rx, ry, rz], a, v)
    movel(p[x_c + -0.044107, y_c + 0.095014, z_c, rx, ry, rz], a, v)
    movel(p[x_c + -0.044075, y_c + 0.095008, z_c, rx, ry, rz], a, v)
    movel(p[x_c + -0.044043, y_c + 0.095002, z_c, rx, ry, rz], a, v)
    movel(p[x_c + -0.044012, y_c + 0.094996, z_c, rx, ry, rz], a, v)
    movel(p[x_c + -0.043981, y_c + 0.094990, z_c, rx, ry, rz], a, v)
    movel(p[x_c + -0.043951, y_c + 0.094985, z_c, rx, ry, rz], a, v)
    movel(p[x_c + -0.043921, y_c + 0.094979, z_c, rx, ry, rz], a, v)
    movel(p[x_c + -0.043891, y_c + 0.094974, z_c, rx, ry, rz], a, v)
    movel(p[x_c + -0.043862, y_c + 0.094969, z_c, rx, ry, rz], a, v)
    movel(p[x_c + -0.043833, y_c + 0.094965, z_c, rx, ry, rz], a, v)
    movel(p[x_c + -0.043804, y_c + 0.094960, z_c, rx, ry, rz], a, v)
    movel(p[x_c + -0.043776, y_c + 0.094956, z_c, rx, ry, rz], a, v)
    movel(p[x_c + -0.043749, y_c + 0.094952, z_c, rx, ry, rz], a, v)
    movel(p[x_c + -0.043722, y_c + 0.094948, z_c, rx, ry, rz], a, v)
    movel(p[x_c + -0.043696, y_c + 0.094945, z_c, rx, ry, rz], a, v)
    movel(p[x_c + -0.043670, y_c + 0.094941, z_c, rx, ry, rz], a, v)
    movel(p[x_c + -0.043645, y_c + 0.094938, z_c, rx, ry, rz], a, v)
    movel(p[x_c + -0.043620, y_c + 0.094936, z_c, rx, ry, rz], a, v)
    movel(p[x_c + -0.043596, y_c + 0.094933, z_c, rx, ry, rz], a, v)
    movel(p[x_c + -0.043573, y_c + 0.094931, z_c, rx, ry, rz], a, v)
    movel(p[x_c + -0.043550, y_c + 0.094929, z_c, rx, ry, rz], a, v)
    movel(p[x_c + -0.043528, y_c + 0.094927, z_c, rx, ry, rz], a, v)
    movel(p[x_c + -0.043507, y_c + 0.094925, z_c, rx, ry, rz], a, v)
    movel(p[x_c + -0.043486, y_c + 0.094924, z_c, rx, ry, rz], a, v)
    movel(p[x_c + -0.043466, y_c + 0.094923, z_c, rx, ry, rz], a, v)
    movel(p[x_c + -0.043447, y_c + 0.094922, z_c, rx, ry, rz], a, v)
    movel(p[x_c + -0.043429, y_c + 0.094921, z_c, rx, ry, rz], a, v)
    movel(p[x_c + -0.043411, y_c + 0.094921, z_c, rx, ry, rz], a, v)
    movel(p[x_c + -0.043394, y_c + 0.094921, z_c, rx, ry, rz], a, v)
    movel(p[x_c + -0.043379, y_c + 0.094921, z_c, rx, ry, rz], a, v)
    movel(p[x_c + -0.043364, y_c + 0.094922, z_c, rx, ry, rz], a, v)
    movel(p[x_c + -0.043349, y_c + 0.094923, z_c, rx, ry, rz], a, v)
    movel(p[x_c + -0.043336, y_c + 0.094924, z_c, rx, ry, rz], a, v)
    movel(p[x_c + -0.043324, y_c + 0.094925, z_c, rx, ry, rz], a, v)
    movel(p[x_c + -0.043312, y_c + 0.094927, z_c, rx, ry, rz], a, v)
    movel(p[x_c + -0.043302, y_c + 0.094928, z_c, rx, ry, rz], a, v)
    movel(p[x_c + -0.043293, y_c + 0.094931, z_c, rx, ry, rz], a, v)
    movel(p[x_c + -0.043284, y_c + 0.094933, z_c, rx, ry, rz], a, v)
    movel(p[x_c + -0.043277, y_c + 0.094936, z_c, rx, ry, rz], a, v)
    movel(p[x_c + -0.043270, y_c + 0.094939, z_c, rx, ry, rz], a, v)
    movel(p[x_c + -0.043265, y_c + 0.094942, z_c, rx, ry, rz], a, v)
    movel(p[x_c + -0.043261, y_c + 0.094946, z_c, rx, ry, rz], a, v)
    movel(p[x_c + -0.043261, y_c + 0.094946, z_c, rx, ry, rz], a, v)
    movel(p[x_c + -0.043250, y_c + 0.094958, z_c, rx, ry, rz], a, v)
    movel(p[x_c + -0.043242, y_c + 0.094970, z_c, rx, ry, rz], a, v)
    movel(p[x_c + -0.043235, y_c + 0.094982, z_c, rx, ry, rz], a, v)
    movel(p[x_c + -0.043231, y_c + 0.094995, z_c, rx, ry, rz], a, v)
    movel(p[x_c + -0.043230, y_c + 0.095008, z_c, rx, ry, rz], a, v)
    movel(p[x_c + -0.043230, y_c + 0.095022, z_c, rx, ry, rz], a, v)
    movel(p[x_c + -0.043233, y_c + 0.095036, z_c, rx, ry, rz], a, v)
    movel(p[x_c + -0.043237, y_c + 0.095050, z_c, rx, ry, rz], a, v)
    movel(p[x_c + -0.043245, y_c + 0.095065, z_c, rx, ry, rz], a, v)
    movel(p[x_c + -0.043254, y_c + 0.095080, z_c, rx, ry, rz], a, v)
    movel(p[x_c + -0.043266, y_c + 0.095096, z_c, rx, ry, rz], a, v)
    movel(p[x_c + -0.043280, y_c + 0.095112, z_c, rx, ry, rz], a, v)
    movel(p[x_c + -0.043297, y_c + 0.095128, z_c, rx, ry, rz], a, v)
    movel(p[x_c + -0.043315, y_c + 0.095145, z_c, rx, ry, rz], a, v)
    movel(p[x_c + -0.043337, y_c + 0.095162, z_c, rx, ry, rz], a, v)
    movel(p[x_c + -0.043360, y_c + 0.095180, z_c, rx, ry, rz], a, v)
    movel(p[x_c + -0.043386, y_c + 0.095198, z_c, rx, ry, rz], a, v)
    movel(p[x_c + -0.043415, y_c + 0.095217, z_c, rx, ry, rz], a, v)
    movel(p[x_c + -0.043446, y_c + 0.095236, z_c, rx, ry, rz], a, v)
    movel(p[x_c + -0.043479, y_c + 0.095256, z_c, rx, ry, rz], a, v)
    movel(p[x_c + -0.043515, y_c + 0.095276, z_c, rx, ry, rz], a, v)
    movel(p[x_c + -0.043553, y_c + 0.095296, z_c, rx, ry, rz], a, v)
    movel(p[x_c + -0.043594, y_c + 0.095317, z_c, rx, ry, rz], a, v)
    movel(p[x_c + -0.043637, y_c + 0.095339, z_c, rx, ry, rz], a, v)
    movel(p[x_c + -0.043683, y_c + 0.095361, z_c, rx, ry, rz], a, v)
    movel(p[x_c + -0.043732, y_c + 0.095384, z_c, rx, ry, rz], a, v)
    movel(p[x_c + -0.043783, y_c + 0.095407, z_c, rx, ry, rz], a, v)
    movel(p[x_c + -0.043837, y_c + 0.095431, z_c, rx, ry, rz], a, v)
    movel(p[x_c + -0.043893, y_c + 0.095455, z_c, rx, ry, rz], a, v)
    movel(p[x_c + -0.043952, y_c + 0.095480, z_c, rx, ry, rz], a, v)
    movel(p[x_c + -0.044013, y_c + 0.095505, z_c, rx, ry, rz], a, v)
    movel(p[x_c + -0.044077, y_c + 0.095531, z_c, rx, ry, rz], a, v)
    movel(p[x_c + -0.044144, y_c + 0.095558, z_c, rx, ry, rz], a, v)
    movel(p[x_c + -0.044214, y_c + 0.095585, z_c, rx, ry, rz], a, v)
    movel(p[x_c + -0.044286, y_c + 0.095613, z_c, rx, ry, rz], a, v)
    movel(p[x_c + -0.044361, y_c + 0.095641, z_c, rx, ry, rz], a, v)
    movel(p[x_c + -0.044439, y_c + 0.095670, z_c, rx, ry, rz], a, v)
    movel(p[x_c + -0.044519, y_c + 0.095700, z_c, rx, ry, rz], a, v)
    movel(p[x_c + -0.044603, y_c + 0.095730, z_c, rx, ry, rz], a, v)
    movel(p[x_c + -0.044689, y_c + 0.095761, z_c, rx, ry, rz], a, v)
    movel(p[x_c + -0.044778, y_c + 0.095793, z_c, rx, ry, rz], a, v)
    movel(p[x_c + -0.044869, y_c + 0.095825, z_c, rx, ry, rz], a, v)
    movel(p[x_c + -0.044964, y_c + 0.095858, z_c, rx, ry, rz], a, v)
    movel(p[x_c + -0.045061, y_c + 0.095892, z_c, rx, ry, rz], a, v)
    movel(p[x_c + -0.045162, y_c + 0.095926, z_c, rx, ry, rz], a, v)
    movel(p[x_c + -0.045265, y_c + 0.095961, z_c, rx, ry, rz], a, v)
    movel(p[x_c + -0.045371, y_c + 0.095997, z_c, rx, ry, rz], a, v)
    movel(p[x_c + -0.045480, y_c + 0.096033, z_c, rx, ry, rz], a, v)
    movel(p[x_c + -0.045592, y_c + 0.096070, z_c, rx, ry, rz], a, v)
    movel(p[x_c + -0.045592, y_c + 0.096070, z_c, rx, ry, rz], a, v)
    movel(p[x_c + -0.045690, y_c + 0.096102, z_c, rx, ry, rz], a, v)
    movel(p[x_c + -0.045785, y_c + 0.096133, z_c, rx, ry, rz], a, v)
    movel(p[x_c + -0.045878, y_c + 0.096163, z_c, rx, ry, rz], a, v)
    movel(p[x_c + -0.045969, y_c + 0.096192, z_c, rx, ry, rz], a, v)
    movel(p[x_c + -0.046058, y_c + 0.096220, z_c, rx, ry, rz], a, v)
    movel(p[x_c + -0.046144, y_c + 0.096246, z_c, rx, ry, rz], a, v)
    movel(p[x_c + -0.046229, y_c + 0.096271, z_c, rx, ry, rz], a, v)
    movel(p[x_c + -0.046313, y_c + 0.096296, z_c, rx, ry, rz], a, v)
    movel(p[x_c + -0.046396, y_c + 0.096319, z_c, rx, ry, rz], a, v)
    movel(p[x_c + -0.046477, y_c + 0.096342, z_c, rx, ry, rz], a, v)
    movel(p[x_c + -0.046558, y_c + 0.096363, z_c, rx, ry, rz], a, v)
    movel(p[x_c + -0.046637, y_c + 0.096383, z_c, rx, ry, rz], a, v)
    movel(p[x_c + -0.046717, y_c + 0.096403, z_c, rx, ry, rz], a, v)
    movel(p[x_c + -0.046796, y_c + 0.096421, z_c, rx, ry, rz], a, v)
    movel(p[x_c + -0.046875, y_c + 0.096439, z_c, rx, ry, rz], a, v)
    movel(p[x_c + -0.046954, y_c + 0.096456, z_c, rx, ry, rz], a, v)
    movel(p[x_c + -0.047034, y_c + 0.096472, z_c, rx, ry, rz], a, v)
    movel(p[x_c + -0.047114, y_c + 0.096487, z_c, rx, ry, rz], a, v)
    movel(p[x_c + -0.047195, y_c + 0.096501, z_c, rx, ry, rz], a, v)
    movel(p[x_c + -0.047277, y_c + 0.096515, z_c, rx, ry, rz], a, v)
    movel(p[x_c + -0.047360, y_c + 0.096528, z_c, rx, ry, rz], a, v)
    movel(p[x_c + -0.047444, y_c + 0.096540, z_c, rx, ry, rz], a, v)
    movel(p[x_c + -0.047530, y_c + 0.096551, z_c, rx, ry, rz], a, v)
    movel(p[x_c + -0.047617, y_c + 0.096562, z_c, rx, ry, rz], a, v)
    movel(p[x_c + -0.047707, y_c + 0.096572, z_c, rx, ry, rz], a, v)
    movel(p[x_c + -0.047798, y_c + 0.096581, z_c, rx, ry, rz], a, v)
    movel(p[x_c + -0.047892, y_c + 0.096590, z_c, rx, ry, rz], a, v)
    movel(p[x_c + -0.047989, y_c + 0.096598, z_c, rx, ry, rz], a, v)
    movel(p[x_c + -0.048088, y_c + 0.096606, z_c, rx, ry, rz], a, v)
    movel(p[x_c + -0.048190, y_c + 0.096612, z_c, rx, ry, rz], a, v)
    movel(p[x_c + -0.048295, y_c + 0.096619, z_c, rx, ry, rz], a, v)
    movel(p[x_c + -0.048404, y_c + 0.096625, z_c, rx, ry, rz], a, v)
    movel(p[x_c + -0.048516, y_c + 0.096630, z_c, rx, ry, rz], a, v)
    movel(p[x_c + -0.048632, y_c + 0.096635, z_c, rx, ry, rz], a, v)
    movel(p[x_c + -0.048751, y_c + 0.096640, z_c, rx, ry, rz], a, v)
    movel(p[x_c + -0.048875, y_c + 0.096644, z_c, rx, ry, rz], a, v)
    movel(p[x_c + -0.049003, y_c + 0.096647, z_c, rx, ry, rz], a, v)
    movel(p[x_c + -0.049136, y_c + 0.096651, z_c, rx, ry, rz], a, v)
    movel(p[x_c + -0.049273, y_c + 0.096654, z_c, rx, ry, rz], a, v)
    movel(p[x_c + -0.049416, y_c + 0.096656, z_c, rx, ry, rz], a, v)
    movel(p[x_c + -0.049563, y_c + 0.096659, z_c, rx, ry, rz], a, v)
    movel(p[x_c + -0.049716, y_c + 0.096661, z_c, rx, ry, rz], a, v)
    movel(p[x_c + -0.049874, y_c + 0.096662, z_c, rx, ry, rz], a, v)
    movel(p[x_c + -0.050038, y_c + 0.096664, z_c, rx, ry, rz], a, v)
    movel(p[x_c + -0.050207, y_c + 0.096665, z_c, rx, ry, rz], a, v)
    movel(p[x_c + -0.050383, y_c + 0.096666, z_c, rx, ry, rz], a, v)
    movel(p[x_c + -0.050566, y_c + 0.096667, z_c, rx, ry, rz], a, v)
    movel(p[x_c + -0.050754, y_c + 0.096668, z_c, rx, ry, rz], a, v)
    movel(p[x_c + -0.050950, y_c + 0.096668, z_c, rx, ry, rz], a, v)
    movel(p[x_c + -0.050950, y_c + 0.096668, z_c, rx, ry, rz], a, v)
    movel(p[x_c + -0.051194, y_c + 0.096668, z_c, rx, ry, rz], a, v)
    movel(p[x_c + -0.051433, y_c + 0.096668, z_c, rx, ry, rz], a, v)
    movel(p[x_c + -0.051667, y_c + 0.096666, z_c, rx, ry, rz], a, v)
    movel(p[x_c + -0.051896, y_c + 0.096664, z_c, rx, ry, rz], a, v)
    movel(p[x_c + -0.052120, y_c + 0.096661, z_c, rx, ry, rz], a, v)
    movel(p[x_c + -0.052340, y_c + 0.096657, z_c, rx, ry, rz], a, v)
    movel(p[x_c + -0.052555, y_c + 0.096652, z_c, rx, ry, rz], a, v)
    movel(p[x_c + -0.052767, y_c + 0.096647, z_c, rx, ry, rz], a, v)
    movel(p[x_c + -0.052975, y_c + 0.096640, z_c, rx, ry, rz], a, v)
    movel(p[x_c + -0.053180, y_c + 0.096632, z_c, rx, ry, rz], a, v)
    movel(p[x_c + -0.053382, y_c + 0.096623, z_c, rx, ry, rz], a, v)
    movel(p[x_c + -0.053581, y_c + 0.096613, z_c, rx, ry, rz], a, v)
    movel(p[x_c + -0.053778, y_c + 0.096601, z_c, rx, ry, rz], a, v)
    movel(p[x_c + -0.053973, y_c + 0.096589, z_c, rx, ry, rz], a, v)
    movel(p[x_c + -0.054166, y_c + 0.096575, z_c, rx, ry, rz], a, v)
    movel(p[x_c + -0.054358, y_c + 0.096560, z_c, rx, ry, rz], a, v)
    movel(p[x_c + -0.054548, y_c + 0.096543, z_c, rx, ry, rz], a, v)
    movel(p[x_c + -0.054738, y_c + 0.096525, z_c, rx, ry, rz], a, v)
    movel(p[x_c + -0.054927, y_c + 0.096506, z_c, rx, ry, rz], a, v)
    movel(p[x_c + -0.055115, y_c + 0.096485, z_c, rx, ry, rz], a, v)
    movel(p[x_c + -0.055304, y_c + 0.096462, z_c, rx, ry, rz], a, v)
    movel(p[x_c + -0.055493, y_c + 0.096438, z_c, rx, ry, rz], a, v)
    movel(p[x_c + -0.055682, y_c + 0.096412, z_c, rx, ry, rz], a, v)
    movel(p[x_c + -0.055872, y_c + 0.096385, z_c, rx, ry, rz], a, v)
    movel(p[x_c + -0.056064, y_c + 0.096355, z_c, rx, ry, rz], a, v)
    movel(p[x_c + -0.056257, y_c + 0.096324, z_c, rx, ry, rz], a, v)
    movel(p[x_c + -0.056451, y_c + 0.096291, z_c, rx, ry, rz], a, v)
    movel(p[x_c + -0.056648, y_c + 0.096257, z_c, rx, ry, rz], a, v)
    movel(p[x_c + -0.056847, y_c + 0.096220, z_c, rx, ry, rz], a, v)
    movel(p[x_c + -0.057049, y_c + 0.096181, z_c, rx, ry, rz], a, v)
    movel(p[x_c + -0.057253, y_c + 0.096140, z_c, rx, ry, rz], a, v)
    movel(p[x_c + -0.057461, y_c + 0.096098, z_c, rx, ry, rz], a, v)
    movel(p[x_c + -0.057672, y_c + 0.096053, z_c, rx, ry, rz], a, v)
    movel(p[x_c + -0.057887, y_c + 0.096006, z_c, rx, ry, rz], a, v)
    movel(p[x_c + -0.058106, y_c + 0.095957, z_c, rx, ry, rz], a, v)
    movel(p[x_c + -0.058330, y_c + 0.095905, z_c, rx, ry, rz], a, v)
    movel(p[x_c + -0.058558, y_c + 0.095851, z_c, rx, ry, rz], a, v)
    movel(p[x_c + -0.058791, y_c + 0.095795, z_c, rx, ry, rz], a, v)
    movel(p[x_c + -0.059030, y_c + 0.095737, z_c, rx, ry, rz], a, v)
    movel(p[x_c + -0.059274, y_c + 0.095676, z_c, rx, ry, rz], a, v)
    movel(p[x_c + -0.059523, y_c + 0.095613, z_c, rx, ry, rz], a, v)
    movel(p[x_c + -0.059779, y_c + 0.095547, z_c, rx, ry, rz], a, v)
    movel(p[x_c + -0.060042, y_c + 0.095478, z_c, rx, ry, rz], a, v)
    movel(p[x_c + -0.060311, y_c + 0.095407, z_c, rx, ry, rz], a, v)
    movel(p[x_c + -0.060587, y_c + 0.095333, z_c, rx, ry, rz], a, v)
    movel(p[x_c + -0.060871, y_c + 0.095257, z_c, rx, ry, rz], a, v)
    movel(p[x_c + -0.061162, y_c + 0.095178, z_c, rx, ry, rz], a, v)
    movel(p[x_c + -0.061461, y_c + 0.095096, z_c, rx, ry, rz], a, v)
    movel(p[x_c + -0.061768, y_c + 0.095011, z_c, rx, ry, rz], a, v)
    movel(p[x_c + -0.061768, y_c + 0.095011, z_c, rx, ry, rz], a, v)
    movel(p[x_c + -0.062033, y_c + 0.094937, z_c, rx, ry, rz], a, v)
    movel(p[x_c + -0.062298, y_c + 0.094862, z_c, rx, ry, rz], a, v)
    movel(p[x_c + -0.062563, y_c + 0.094786, z_c, rx, ry, rz], a, v)
    movel(p[x_c + -0.062828, y_c + 0.094709, z_c, rx, ry, rz], a, v)
    movel(p[x_c + -0.063093, y_c + 0.094631, z_c, rx, ry, rz], a, v)
    movel(p[x_c + -0.063357, y_c + 0.094552, z_c, rx, ry, rz], a, v)
    movel(p[x_c + -0.063621, y_c + 0.094472, z_c, rx, ry, rz], a, v)
    movel(p[x_c + -0.063885, y_c + 0.094391, z_c, rx, ry, rz], a, v)
    movel(p[x_c + -0.064149, y_c + 0.094309, z_c, rx, ry, rz], a, v)
    movel(p[x_c + -0.064412, y_c + 0.094226, z_c, rx, ry, rz], a, v)
    movel(p[x_c + -0.064674, y_c + 0.094142, z_c, rx, ry, rz], a, v)
    movel(p[x_c + -0.064937, y_c + 0.094058, z_c, rx, ry, rz], a, v)
    movel(p[x_c + -0.065199, y_c + 0.093972, z_c, rx, ry, rz], a, v)
    movel(p[x_c + -0.065460, y_c + 0.093885, z_c, rx, ry, rz], a, v)
    movel(p[x_c + -0.065721, y_c + 0.093798, z_c, rx, ry, rz], a, v)
    movel(p[x_c + -0.065982, y_c + 0.093709, z_c, rx, ry, rz], a, v)
    movel(p[x_c + -0.066242, y_c + 0.093620, z_c, rx, ry, rz], a, v)
    movel(p[x_c + -0.066502, y_c + 0.093530, z_c, rx, ry, rz], a, v)
    movel(p[x_c + -0.066761, y_c + 0.093439, z_c, rx, ry, rz], a, v)
    movel(p[x_c + -0.067019, y_c + 0.093347, z_c, rx, ry, rz], a, v)
    movel(p[x_c + -0.067277, y_c + 0.093254, z_c, rx, ry, rz], a, v)
    movel(p[x_c + -0.067535, y_c + 0.093161, z_c, rx, ry, rz], a, v)
    movel(p[x_c + -0.067791, y_c + 0.093066, z_c, rx, ry, rz], a, v)
    movel(p[x_c + -0.068047, y_c + 0.092971, z_c, rx, ry, rz], a, v)
    movel(p[x_c + -0.068303, y_c + 0.092875, z_c, rx, ry, rz], a, v)
    movel(p[x_c + -0.068557, y_c + 0.092778, z_c, rx, ry, rz], a, v)
    movel(p[x_c + -0.068811, y_c + 0.092680, z_c, rx, ry, rz], a, v)
    movel(p[x_c + -0.069064, y_c + 0.092581, z_c, rx, ry, rz], a, v)
    movel(p[x_c + -0.069317, y_c + 0.092482, z_c, rx, ry, rz], a, v)
    movel(p[x_c + -0.069568, y_c + 0.092382, z_c, rx, ry, rz], a, v)
    movel(p[x_c + -0.069819, y_c + 0.092281, z_c, rx, ry, rz], a, v)
    movel(p[x_c + -0.070069, y_c + 0.092179, z_c, rx, ry, rz], a, v)
    movel(p[x_c + -0.070318, y_c + 0.092077, z_c, rx, ry, rz], a, v)
    movel(p[x_c + -0.070566, y_c + 0.091974, z_c, rx, ry, rz], a, v)
    movel(p[x_c + -0.070813, y_c + 0.091870, z_c, rx, ry, rz], a, v)
    movel(p[x_c + -0.071060, y_c + 0.091765, z_c, rx, ry, rz], a, v)
    movel(p[x_c + -0.071305, y_c + 0.091660, z_c, rx, ry, rz], a, v)
    movel(p[x_c + -0.071549, y_c + 0.091554, z_c, rx, ry, rz], a, v)
    movel(p[x_c + -0.071793, y_c + 0.091447, z_c, rx, ry, rz], a, v)
    movel(p[x_c + -0.072035, y_c + 0.091340, z_c, rx, ry, rz], a, v)
    movel(p[x_c + -0.072276, y_c + 0.091231, z_c, rx, ry, rz], a, v)
    movel(p[x_c + -0.072516, y_c + 0.091123, z_c, rx, ry, rz], a, v)
    movel(p[x_c + -0.072756, y_c + 0.091013, z_c, rx, ry, rz], a, v)
    movel(p[x_c + -0.072994, y_c + 0.090903, z_c, rx, ry, rz], a, v)
    movel(p[x_c + -0.073230, y_c + 0.090792, z_c, rx, ry, rz], a, v)
    movel(p[x_c + -0.073466, y_c + 0.090681, z_c, rx, ry, rz], a, v)
    movel(p[x_c + -0.073701, y_c + 0.090569, z_c, rx, ry, rz], a, v)
    movel(p[x_c + -0.073934, y_c + 0.090456, z_c, rx, ry, rz], a, v)
    movel(p[x_c + -0.074166, y_c + 0.090343, z_c, rx, ry, rz], a, v)
    movel(p[x_c + -0.074166, y_c + 0.090343, z_c, rx, ry, rz], a, v)
    movel(p[x_c + -0.074335, y_c + 0.090260, z_c, rx, ry, rz], a, v)
    movel(p[x_c + -0.074502, y_c + 0.090177, z_c, rx, ry, rz], a, v)
    movel(p[x_c + -0.074666, y_c + 0.090096, z_c, rx, ry, rz], a, v)
    movel(p[x_c + -0.074827, y_c + 0.090015, z_c, rx, ry, rz], a, v)
    movel(p[x_c + -0.074986, y_c + 0.089935, z_c, rx, ry, rz], a, v)
    movel(p[x_c + -0.075142, y_c + 0.089856, z_c, rx, ry, rz], a, v)
    movel(p[x_c + -0.075295, y_c + 0.089778, z_c, rx, ry, rz], a, v)
    movel(p[x_c + -0.075445, y_c + 0.089701, z_c, rx, ry, rz], a, v)
    movel(p[x_c + -0.075592, y_c + 0.089626, z_c, rx, ry, rz], a, v)
    movel(p[x_c + -0.075736, y_c + 0.089551, z_c, rx, ry, rz], a, v)
    movel(p[x_c + -0.075877, y_c + 0.089478, z_c, rx, ry, rz], a, v)
    movel(p[x_c + -0.076014, y_c + 0.089406, z_c, rx, ry, rz], a, v)
    movel(p[x_c + -0.076148, y_c + 0.089336, z_c, rx, ry, rz], a, v)
    movel(p[x_c + -0.076278, y_c + 0.089267, z_c, rx, ry, rz], a, v)
    movel(p[x_c + -0.076404, y_c + 0.089199, z_c, rx, ry, rz], a, v)
    movel(p[x_c + -0.076527, y_c + 0.089133, z_c, rx, ry, rz], a, v)
    movel(p[x_c + -0.076646, y_c + 0.089068, z_c, rx, ry, rz], a, v)
    movel(p[x_c + -0.076761, y_c + 0.089005, z_c, rx, ry, rz], a, v)
    movel(p[x_c + -0.076872, y_c + 0.088944, z_c, rx, ry, rz], a, v)
    movel(p[x_c + -0.076979, y_c + 0.088885, z_c, rx, ry, rz], a, v)
    movel(p[x_c + -0.077081, y_c + 0.088827, z_c, rx, ry, rz], a, v)
    movel(p[x_c + -0.077179, y_c + 0.088772, z_c, rx, ry, rz], a, v)
    movel(p[x_c + -0.077273, y_c + 0.088718, z_c, rx, ry, rz], a, v)
    movel(p[x_c + -0.077362, y_c + 0.088666, z_c, rx, ry, rz], a, v)
    movel(p[x_c + -0.077447, y_c + 0.088616, z_c, rx, ry, rz], a, v)
    movel(p[x_c + -0.077527, y_c + 0.088569, z_c, rx, ry, rz], a, v)
    movel(p[x_c + -0.077602, y_c + 0.088523, z_c, rx, ry, rz], a, v)
    movel(p[x_c + -0.077673, y_c + 0.088480, z_c, rx, ry, rz], a, v)
    movel(p[x_c + -0.077738, y_c + 0.088439, z_c, rx, ry, rz], a, v)
    movel(p[x_c + -0.077798, y_c + 0.088400, z_c, rx, ry, rz], a, v)
    movel(p[x_c + -0.077853, y_c + 0.088363, z_c, rx, ry, rz], a, v)
    movel(p[x_c + -0.077903, y_c + 0.088329, z_c, rx, ry, rz], a, v)
    movel(p[x_c + -0.077947, y_c + 0.088298, z_c, rx, ry, rz], a, v)
    movel(p[x_c + -0.077986, y_c + 0.088269, z_c, rx, ry, rz], a, v)
    movel(p[x_c + -0.078019, y_c + 0.088243, z_c, rx, ry, rz], a, v)
    movel(p[x_c + -0.078047, y_c + 0.088219, z_c, rx, ry, rz], a, v)
    movel(p[x_c + -0.078069, y_c + 0.088198, z_c, rx, ry, rz], a, v)
    movel(p[x_c + -0.078085, y_c + 0.088180, z_c, rx, ry, rz], a, v)
    movel(p[x_c + -0.078095, y_c + 0.088164, z_c, rx, ry, rz], a, v)
    movel(p[x_c + -0.078099, y_c + 0.088152, z_c, rx, ry, rz], a, v)
    movel(p[x_c + -0.078097, y_c + 0.088142, z_c, rx, ry, rz], a, v)
    movel(p[x_c + -0.078089, y_c + 0.088136, z_c, rx, ry, rz], a, v)
    movel(p[x_c + -0.078074, y_c + 0.088132, z_c, rx, ry, rz], a, v)
    movel(p[x_c + -0.078053, y_c + 0.088131, z_c, rx, ry, rz], a, v)
    movel(p[x_c + -0.078026, y_c + 0.088134, z_c, rx, ry, rz], a, v)
    movel(p[x_c + -0.077992, y_c + 0.088140, z_c, rx, ry, rz], a, v)
    movel(p[x_c + -0.077951, y_c + 0.088149, z_c, rx, ry, rz], a, v)
    movel(p[x_c + -0.077903, y_c + 0.088162, z_c, rx, ry, rz], a, v)
    movel(p[x_c + -0.077849, y_c + 0.088177, z_c, rx, ry, rz], a, v)
    movel(p[x_c + -0.077849, y_c + 0.088177, z_c, rx, ry, rz], a, v)
    movel(p[x_c + -0.077835, y_c + 0.088182, z_c, rx, ry, rz], a, v)
    movel(p[x_c + -0.077816, y_c + 0.088188, z_c, rx, ry, rz], a, v)
    movel(p[x_c + -0.077793, y_c + 0.088195, z_c, rx, ry, rz], a, v)
    movel(p[x_c + -0.077764, y_c + 0.088204, z_c, rx, ry, rz], a, v)
    movel(p[x_c + -0.077731, y_c + 0.088215, z_c, rx, ry, rz], a, v)
    movel(p[x_c + -0.077694, y_c + 0.088227, z_c, rx, ry, rz], a, v)
    movel(p[x_c + -0.077651, y_c + 0.088241, z_c, rx, ry, rz], a, v)
    movel(p[x_c + -0.077605, y_c + 0.088256, z_c, rx, ry, rz], a, v)
    movel(p[x_c + -0.077554, y_c + 0.088272, z_c, rx, ry, rz], a, v)
    movel(p[x_c + -0.077499, y_c + 0.088290, z_c, rx, ry, rz], a, v)
    movel(p[x_c + -0.077439, y_c + 0.088309, z_c, rx, ry, rz], a, v)
    movel(p[x_c + -0.077376, y_c + 0.088330, z_c, rx, ry, rz], a, v)
    movel(p[x_c + -0.077308, y_c + 0.088351, z_c, rx, ry, rz], a, v)
    movel(p[x_c + -0.077237, y_c + 0.088375, z_c, rx, ry, rz], a, v)
    movel(p[x_c + -0.077162, y_c + 0.088399, z_c, rx, ry, rz], a, v)
    movel(p[x_c + -0.077083, y_c + 0.088425, z_c, rx, ry, rz], a, v)
    movel(p[x_c + -0.077000, y_c + 0.088451, z_c, rx, ry, rz], a, v)
    movel(p[x_c + -0.076914, y_c + 0.088479, z_c, rx, ry, rz], a, v)
    movel(p[x_c + -0.076825, y_c + 0.088508, z_c, rx, ry, rz], a, v)
    movel(p[x_c + -0.076732, y_c + 0.088539, z_c, rx, ry, rz], a, v)
    movel(p[x_c + -0.076636, y_c + 0.088570, z_c, rx, ry, rz], a, v)
    movel(p[x_c + -0.076536, y_c + 0.088602, z_c, rx, ry, rz], a, v)
    movel(p[x_c + -0.076434, y_c + 0.088635, z_c, rx, ry, rz], a, v)
    movel(p[x_c + -0.076328, y_c + 0.088670, z_c, rx, ry, rz], a, v)
    movel(p[x_c + -0.076219, y_c + 0.088705, z_c, rx, ry, rz], a, v)
    movel(p[x_c + -0.076108, y_c + 0.088741, z_c, rx, ry, rz], a, v)
    movel(p[x_c + -0.075994, y_c + 0.088779, z_c, rx, ry, rz], a, v)
    movel(p[x_c + -0.075877, y_c + 0.088817, z_c, rx, ry, rz], a, v)
    movel(p[x_c + -0.075757, y_c + 0.088855, z_c, rx, ry, rz], a, v)
    movel(p[x_c + -0.075635, y_c + 0.088895, z_c, rx, ry, rz], a, v)
    movel(p[x_c + -0.075511, y_c + 0.088936, z_c, rx, ry, rz], a, v)
    movel(p[x_c + -0.075384, y_c + 0.088977, z_c, rx, ry, rz], a, v)
    movel(p[x_c + -0.075255, y_c + 0.089019, z_c, rx, ry, rz], a, v)
    movel(p[x_c + -0.075124, y_c + 0.089062, z_c, rx, ry, rz], a, v)
    movel(p[x_c + -0.074991, y_c + 0.089105, z_c, rx, ry, rz], a, v)
    movel(p[x_c + -0.074856, y_c + 0.089149, z_c, rx, ry, rz], a, v)
    movel(p[x_c + -0.074719, y_c + 0.089194, z_c, rx, ry, rz], a, v)
    movel(p[x_c + -0.074580, y_c + 0.089239, z_c, rx, ry, rz], a, v)
    movel(p[x_c + -0.074439, y_c + 0.089285, z_c, rx, ry, rz], a, v)
    movel(p[x_c + -0.074297, y_c + 0.089332, z_c, rx, ry, rz], a, v)
    movel(p[x_c + -0.074153, y_c + 0.089379, z_c, rx, ry, rz], a, v)
    movel(p[x_c + -0.074008, y_c + 0.089426, z_c, rx, ry, rz], a, v)
    movel(p[x_c + -0.073861, y_c + 0.089474, z_c, rx, ry, rz], a, v)
    movel(p[x_c + -0.073713, y_c + 0.089522, z_c, rx, ry, rz], a, v)
    movel(p[x_c + -0.073564, y_c + 0.089571, z_c, rx, ry, rz], a, v)
    movel(p[x_c + -0.073414, y_c + 0.089620, z_c, rx, ry, rz], a, v)
    movel(p[x_c + -0.073263, y_c + 0.089670, z_c, rx, ry, rz], a, v)
    movel(p[x_c + -0.073110, y_c + 0.089719, z_c, rx, ry, rz], a, v)
    movel(p[x_c + -0.072957, y_c + 0.089770, z_c, rx, ry, rz], a, v)
    movel(p[x_c + -0.072957, y_c + 0.089770, z_c, rx, ry, rz], a, v)
    movel(p[x_c + -0.072957, y_c + 0.089770, z_c, rx, ry, rz], a, v)
    movel(p[x_c + -0.072957, y_c + 0.089770, z_c, rx, ry, rz], a, v)
    movel(p[x_c + -0.072957, y_c + 0.089770, z_c, rx, ry, rz], a, v)
    movel(p[x_c + -0.072957, y_c + 0.089770, z_c, rx, ry, rz], a, v)
    movel(p[x_c + -0.072957, y_c + 0.089770, z_c, rx, ry, rz], a, v)
    movel(p[x_c + -0.072957, y_c + 0.089770, z_c, rx, ry, rz], a, v)
    movel(p[x_c + -0.072957, y_c + 0.089770, z_c, rx, ry, rz], a, v)
    movel(p[x_c + -0.072957, y_c + 0.089770, z_c, rx, ry, rz], a, v)
    movel(p[x_c + -0.072957, y_c + 0.089770, z_c, rx, ry, rz], a, v)
    movel(p[x_c + -0.031735, y_c + 0.100277, z_c, rx, ry, rz], a, v)
    movel(p[x_c + -0.031735, y_c + 0.100277, z_c, rx, ry, rz], a, v)
    movel(p[x_c + -0.031735, y_c + 0.100277, z_c, rx, ry, rz], a, v)
    movel(p[x_c + -0.031735, y_c + 0.100277, z_c, rx, ry, rz], a, v)
    movel(p[x_c + -0.031735, y_c + 0.100277, z_c, rx, ry, rz], a, v)
    movel(p[x_c + -0.031735, y_c + 0.100277, z_c, rx, ry, rz], a, v)
    movel(p[x_c + -0.031735, y_c + 0.100277, z_c, rx, ry, rz], a, v)
    movel(p[x_c + -0.031735, y_c + 0.100277, z_c, rx, ry, rz], a, v)
    movel(p[x_c + -0.031735, y_c + 0.100277, z_c, rx, ry, rz], a, v)
    movel(p[x_c + -0.031735, y_c + 0.100277, z_c, rx, ry, rz], a, v)
    movel(p[x_c + -0.031735, y_c + 0.100277, z_c, rx, ry, rz], a, v)
    movel(p[x_c + -0.031684, y_c + 0.100302, z_c, rx, ry, rz], a, v)
    movel(p[x_c + -0.031634, y_c + 0.100328, z_c, rx, ry, rz], a, v)
    movel(p[x_c + -0.031582, y_c + 0.100355, z_c, rx, ry, rz], a, v)
    movel(p[x_c + -0.031531, y_c + 0.100384, z_c, rx, ry, rz], a, v)
    movel(p[x_c + -0.031479, y_c + 0.100413, z_c, rx, ry, rz], a, v)
    movel(p[x_c + -0.031427, y_c + 0.100443, z_c, rx, ry, rz], a, v)
    movel(p[x_c + -0.031374, y_c + 0.100474, z_c, rx, ry, rz], a, v)
    movel(p[x_c + -0.031321, y_c + 0.100506, z_c, rx, ry, rz], a, v)
    movel(p[x_c + -0.031268, y_c + 0.100539, z_c, rx, ry, rz], a, v)
    movel(p[x_c + -0.031214, y_c + 0.100574, z_c, rx, ry, rz], a, v)
    movel(p[x_c + -0.031160, y_c + 0.100609, z_c, rx, ry, rz], a, v)
    movel(p[x_c + -0.031106, y_c + 0.100645, z_c, rx, ry, rz], a, v)
    movel(p[x_c + -0.031051, y_c + 0.100683, z_c, rx, ry, rz], a, v)
    movel(p[x_c + -0.030996, y_c + 0.100721, z_c, rx, ry, rz], a, v)
    movel(p[x_c + -0.030940, y_c + 0.100761, z_c, rx, ry, rz], a, v)
    movel(p[x_c + -0.030884, y_c + 0.100802, z_c, rx, ry, rz], a, v)
    movel(p[x_c + -0.030828, y_c + 0.100843, z_c, rx, ry, rz], a, v)
    movel(p[x_c + -0.030771, y_c + 0.100886, z_c, rx, ry, rz], a, v)
    movel(p[x_c + -0.030713, y_c + 0.100930, z_c, rx, ry, rz], a, v)
    movel(p[x_c + -0.030655, y_c + 0.100975, z_c, rx, ry, rz], a, v)
    movel(p[x_c + -0.030597, y_c + 0.101022, z_c, rx, ry, rz], a, v)
    movel(p[x_c + -0.030538, y_c + 0.101069, z_c, rx, ry, rz], a, v)
    movel(p[x_c + -0.030479, y_c + 0.101117, z_c, rx, ry, rz], a, v)
    movel(p[x_c + -0.030419, y_c + 0.101167, z_c, rx, ry, rz], a, v)
    movel(p[x_c + -0.030359, y_c + 0.101218, z_c, rx, ry, rz], a, v)
    movel(p[x_c + -0.030298, y_c + 0.101270, z_c, rx, ry, rz], a, v)
    movel(p[x_c + -0.030236, y_c + 0.101323, z_c, rx, ry, rz], a, v)
    movel(p[x_c + -0.030175, y_c + 0.101377, z_c, rx, ry, rz], a, v)
    movel(p[x_c + -0.030112, y_c + 0.101433, z_c, rx, ry, rz], a, v)
    movel(p[x_c + -0.030049, y_c + 0.101489, z_c, rx, ry, rz], a, v)
    movel(p[x_c + -0.029985, y_c + 0.101547, z_c, rx, ry, rz], a, v)
    movel(p[x_c + -0.029921, y_c + 0.101606, z_c, rx, ry, rz], a, v)
    movel(p[x_c + -0.029857, y_c + 0.101667, z_c, rx, ry, rz], a, v)
    movel(p[x_c + -0.029791, y_c + 0.101728, z_c, rx, ry, rz], a, v)
    movel(p[x_c + -0.029725, y_c + 0.101791, z_c, rx, ry, rz], a, v)
    movel(p[x_c + -0.029659, y_c + 0.101855, z_c, rx, ry, rz], a, v)
    movel(p[x_c + -0.029592, y_c + 0.101920, z_c, rx, ry, rz], a, v)
    movel(p[x_c + -0.029524, y_c + 0.101987, z_c, rx, ry, rz], a, v)
    movel(p[x_c + -0.029455, y_c + 0.102055, z_c, rx, ry, rz], a, v)
    movel(p[x_c + -0.029386, y_c + 0.102124, z_c, rx, ry, rz], a, v)
    movel(p[x_c + -0.029317, y_c + 0.102194, z_c, rx, ry, rz], a, v)
    movel(p[x_c + -0.029246, y_c + 0.102266, z_c, rx, ry, rz], a, v)
    movel(p[x_c + -0.029175, y_c + 0.102339, z_c, rx, ry, rz], a, v)
    movel(p[x_c + -0.029104, y_c + 0.102413, z_c, rx, ry, rz], a, v)
    movel(p[x_c + -0.029031, y_c + 0.102488, z_c, rx, ry, rz], a, v)
    movel(p[x_c + -0.028958, y_c + 0.102565, z_c, rx, ry, rz], a, v)
    movel(p[x_c + -0.028884, y_c + 0.102643, z_c, rx, ry, rz], a, v)
    movel(p[x_c + -0.028810, y_c + 0.102723, z_c, rx, ry, rz], a, v)
    movel(p[x_c + -0.028734, y_c + 0.102804, z_c, rx, ry, rz], a, v)
    movel(p[x_c + -0.028734, y_c + 0.102804, z_c, rx, ry, rz], a, v)
    movel(p[x_c + -0.026935, y_c + 0.104743, z_c, rx, ry, rz], a, v)
    movel(p[x_c + -0.026935, y_c + 0.104743, z_c, rx, ry, rz], a, v)
    movel(p[x_c + -0.027867, y_c + 0.105017, z_c, rx, ry, rz], a, v)
    movel(p[x_c + -0.027867, y_c + 0.105017, z_c, rx, ry, rz], a, v)
    movel(p[x_c + -0.028120, y_c + 0.105090, z_c, rx, ry, rz], a, v)
    movel(p[x_c + -0.028369, y_c + 0.105157, z_c, rx, ry, rz], a, v)
    movel(p[x_c + -0.028614, y_c + 0.105220, z_c, rx, ry, rz], a, v)
    movel(p[x_c + -0.028857, y_c + 0.105278, z_c, rx, ry, rz], a, v)
    movel(p[x_c + -0.029096, y_c + 0.105332, z_c, rx, ry, rz], a, v)
    movel(p[x_c + -0.029333, y_c + 0.105381, z_c, rx, ry, rz], a, v)
    movel(p[x_c + -0.029566, y_c + 0.105425, z_c, rx, ry, rz], a, v)
    movel(p[x_c + -0.029798, y_c + 0.105464, z_c, rx, ry, rz], a, v)
    movel(p[x_c + -0.030026, y_c + 0.105498, z_c, rx, ry, rz], a, v)
    movel(p[x_c + -0.030253, y_c + 0.105527, z_c, rx, ry, rz], a, v)
    movel(p[x_c + -0.030477, y_c + 0.105552, z_c, rx, ry, rz], a, v)
    movel(p[x_c + -0.030699, y_c + 0.105571, z_c, rx, ry, rz], a, v)
    movel(p[x_c + -0.030920, y_c + 0.105586, z_c, rx, ry, rz], a, v)
    movel(p[x_c + -0.031139, y_c + 0.105595, z_c, rx, ry, rz], a, v)
    movel(p[x_c + -0.031356, y_c + 0.105599, z_c, rx, ry, rz], a, v)
    movel(p[x_c + -0.031572, y_c + 0.105598, z_c, rx, ry, rz], a, v)
    movel(p[x_c + -0.031786, y_c + 0.105592, z_c, rx, ry, rz], a, v)
    movel(p[x_c + -0.032000, y_c + 0.105581, z_c, rx, ry, rz], a, v)
    movel(p[x_c + -0.032212, y_c + 0.105565, z_c, rx, ry, rz], a, v)
    movel(p[x_c + -0.032424, y_c + 0.105543, z_c, rx, ry, rz], a, v)
    movel(p[x_c + -0.032634, y_c + 0.105516, z_c, rx, ry, rz], a, v)
    movel(p[x_c + -0.032845, y_c + 0.105484, z_c, rx, ry, rz], a, v)
    movel(p[x_c + -0.033055, y_c + 0.105446, z_c, rx, ry, rz], a, v)
    movel(p[x_c + -0.033265, y_c + 0.105403, z_c, rx, ry, rz], a, v)
    movel(p[x_c + -0.033474, y_c + 0.105355, z_c, rx, ry, rz], a, v)
    movel(p[x_c + -0.033684, y_c + 0.105301, z_c, rx, ry, rz], a, v)
    movel(p[x_c + -0.033894, y_c + 0.105242, z_c, rx, ry, rz], a, v)
    movel(p[x_c + -0.034104, y_c + 0.105177, z_c, rx, ry, rz], a, v)
    movel(p[x_c + -0.034315, y_c + 0.105107, z_c, rx, ry, rz], a, v)
    movel(p[x_c + -0.034526, y_c + 0.105031, z_c, rx, ry, rz], a, v)
    movel(p[x_c + -0.034738, y_c + 0.104949, z_c, rx, ry, rz], a, v)
    movel(p[x_c + -0.034951, y_c + 0.104862, z_c, rx, ry, rz], a, v)
    movel(p[x_c + -0.035165, y_c + 0.104769, z_c, rx, ry, rz], a, v)
    movel(p[x_c + -0.035381, y_c + 0.104670, z_c, rx, ry, rz], a, v)
    movel(p[x_c + -0.035597, y_c + 0.104566, z_c, rx, ry, rz], a, v)
    movel(p[x_c + -0.035816, y_c + 0.104455, z_c, rx, ry, rz], a, v)
    movel(p[x_c + -0.036036, y_c + 0.104339, z_c, rx, ry, rz], a, v)
    movel(p[x_c + -0.036257, y_c + 0.104217, z_c, rx, ry, rz], a, v)
    movel(p[x_c + -0.036481, y_c + 0.104089, z_c, rx, ry, rz], a, v)
    movel(p[x_c + -0.036707, y_c + 0.103956, z_c, rx, ry, rz], a, v)
    movel(p[x_c + -0.036935, y_c + 0.103816, z_c, rx, ry, rz], a, v)
    movel(p[x_c + -0.037165, y_c + 0.103670, z_c, rx, ry, rz], a, v)
    movel(p[x_c + -0.037398, y_c + 0.103519, z_c, rx, ry, rz], a, v)
    movel(p[x_c + -0.037634, y_c + 0.103361, z_c, rx, ry, rz], a, v)
    movel(p[x_c + -0.037872, y_c + 0.103197, z_c, rx, ry, rz], a, v)
    movel(p[x_c + -0.038114, y_c + 0.103027, z_c, rx, ry, rz], a, v)
    movel(p[x_c + -0.038358, y_c + 0.102851, z_c, rx, ry, rz], a, v)
    movel(p[x_c + -0.038606, y_c + 0.102668, z_c, rx, ry, rz], a, v)
    movel(p[x_c + -0.038857, y_c + 0.102480, z_c, rx, ry, rz], a, v)
    movel(p[x_c + -0.038857, y_c + 0.102480, z_c, rx, ry, rz], a, v)
    movel(p[x_c + -0.038948, y_c + 0.102411, z_c, rx, ry, rz], a, v)
    movel(p[x_c + -0.039036, y_c + 0.102344, z_c, rx, ry, rz], a, v)
    movel(p[x_c + -0.039121, y_c + 0.102278, z_c, rx, ry, rz], a, v)
    movel(p[x_c + -0.039204, y_c + 0.102215, z_c, rx, ry, rz], a, v)
    movel(p[x_c + -0.039284, y_c + 0.102153, z_c, rx, ry, rz], a, v)
    movel(p[x_c + -0.039361, y_c + 0.102093, z_c, rx, ry, rz], a, v)
    movel(p[x_c + -0.039436, y_c + 0.102035, z_c, rx, ry, rz], a, v)
    movel(p[x_c + -0.039507, y_c + 0.101978, z_c, rx, ry, rz], a, v)
    movel(p[x_c + -0.039577, y_c + 0.101923, z_c, rx, ry, rz], a, v)
    movel(p[x_c + -0.039644, y_c + 0.101870, z_c, rx, ry, rz], a, v)
    movel(p[x_c + -0.039708, y_c + 0.101818, z_c, rx, ry, rz], a, v)
    movel(p[x_c + -0.039769, y_c + 0.101768, z_c, rx, ry, rz], a, v)
    movel(p[x_c + -0.039828, y_c + 0.101719, z_c, rx, ry, rz], a, v)
    movel(p[x_c + -0.039885, y_c + 0.101672, z_c, rx, ry, rz], a, v)
    movel(p[x_c + -0.039939, y_c + 0.101627, z_c, rx, ry, rz], a, v)
    movel(p[x_c + -0.039991, y_c + 0.101583, z_c, rx, ry, rz], a, v)
    movel(p[x_c + -0.040040, y_c + 0.101540, z_c, rx, ry, rz], a, v)
    movel(p[x_c + -0.040087, y_c + 0.101499, z_c, rx, ry, rz], a, v)
    movel(p[x_c + -0.040132, y_c + 0.101459, z_c, rx, ry, rz], a, v)
    movel(p[x_c + -0.040174, y_c + 0.101421, z_c, rx, ry, rz], a, v)
    movel(p[x_c + -0.040214, y_c + 0.101384, z_c, rx, ry, rz], a, v)
    movel(p[x_c + -0.040252, y_c + 0.101348, z_c, rx, ry, rz], a, v)
    movel(p[x_c + -0.040287, y_c + 0.101314, z_c, rx, ry, rz], a, v)
    movel(p[x_c + -0.040320, y_c + 0.101281, z_c, rx, ry, rz], a, v)
    movel(p[x_c + -0.040351, y_c + 0.101249, z_c, rx, ry, rz], a, v)
    movel(p[x_c + -0.040380, y_c + 0.101218, z_c, rx, ry, rz], a, v)
    movel(p[x_c + -0.040407, y_c + 0.101189, z_c, rx, ry, rz], a, v)
    movel(p[x_c + -0.040431, y_c + 0.101161, z_c, rx, ry, rz], a, v)
    movel(p[x_c + -0.040453, y_c + 0.101134, z_c, rx, ry, rz], a, v)
    movel(p[x_c + -0.040474, y_c + 0.101108, z_c, rx, ry, rz], a, v)
    movel(p[x_c + -0.040492, y_c + 0.101083, z_c, rx, ry, rz], a, v)
    movel(p[x_c + -0.040508, y_c + 0.101060, z_c, rx, ry, rz], a, v)
    movel(p[x_c + -0.040522, y_c + 0.101037, z_c, rx, ry, rz], a, v)
    movel(p[x_c + -0.040534, y_c + 0.101016, z_c, rx, ry, rz], a, v)
    movel(p[x_c + -0.040544, y_c + 0.100995, z_c, rx, ry, rz], a, v)
    movel(p[x_c + -0.040553, y_c + 0.100975, z_c, rx, ry, rz], a, v)
    movel(p[x_c + -0.040559, y_c + 0.100957, z_c, rx, ry, rz], a, v)
    movel(p[x_c + -0.040563, y_c + 0.100939, z_c, rx, ry, rz], a, v)
    movel(p[x_c + -0.040566, y_c + 0.100922, z_c, rx, ry, rz], a, v)
    movel(p[x_c + -0.040566, y_c + 0.100906, z_c, rx, ry, rz], a, v)
    movel(p[x_c + -0.040565, y_c + 0.100891, z_c, rx, ry, rz], a, v)
    movel(p[x_c + -0.040562, y_c + 0.100877, z_c, rx, ry, rz], a, v)
    movel(p[x_c + -0.040558, y_c + 0.100864, z_c, rx, ry, rz], a, v)
    movel(p[x_c + -0.040551, y_c + 0.100851, z_c, rx, ry, rz], a, v)
    movel(p[x_c + -0.040543, y_c + 0.100839, z_c, rx, ry, rz], a, v)
    movel(p[x_c + -0.040533, y_c + 0.100828, z_c, rx, ry, rz], a, v)
    movel(p[x_c + -0.040522, y_c + 0.100818, z_c, rx, ry, rz], a, v)
    movel(p[x_c + -0.040508, y_c + 0.100808, z_c, rx, ry, rz], a, v)
    movel(p[x_c + -0.040493, y_c + 0.100799, z_c, rx, ry, rz], a, v)
    movel(p[x_c + -0.040493, y_c + 0.100799, z_c, rx, ry, rz], a, v)
    movel(p[x_c + -0.040481, y_c + 0.100792, z_c, rx, ry, rz], a, v)
    movel(p[x_c + -0.040467, y_c + 0.100785, z_c, rx, ry, rz], a, v)
    movel(p[x_c + -0.040450, y_c + 0.100778, z_c, rx, ry, rz], a, v)
    movel(p[x_c + -0.040432, y_c + 0.100769, z_c, rx, ry, rz], a, v)
    movel(p[x_c + -0.040411, y_c + 0.100761, z_c, rx, ry, rz], a, v)
    movel(p[x_c + -0.040389, y_c + 0.100751, z_c, rx, ry, rz], a, v)
    movel(p[x_c + -0.040365, y_c + 0.100741, z_c, rx, ry, rz], a, v)
    movel(p[x_c + -0.040339, y_c + 0.100731, z_c, rx, ry, rz], a, v)
    movel(p[x_c + -0.040311, y_c + 0.100720, z_c, rx, ry, rz], a, v)
    movel(p[x_c + -0.040281, y_c + 0.100709, z_c, rx, ry, rz], a, v)
    movel(p[x_c + -0.040250, y_c + 0.100698, z_c, rx, ry, rz], a, v)
    movel(p[x_c + -0.040217, y_c + 0.100686, z_c, rx, ry, rz], a, v)
    movel(p[x_c + -0.040182, y_c + 0.100673, z_c, rx, ry, rz], a, v)
    movel(p[x_c + -0.040146, y_c + 0.100660, z_c, rx, ry, rz], a, v)
    movel(p[x_c + -0.040108, y_c + 0.100647, z_c, rx, ry, rz], a, v)
    movel(p[x_c + -0.040069, y_c + 0.100633, z_c, rx, ry, rz], a, v)
    movel(p[x_c + -0.040028, y_c + 0.100619, z_c, rx, ry, rz], a, v)
    movel(p[x_c + -0.039985, y_c + 0.100605, z_c, rx, ry, rz], a, v)
    movel(p[x_c + -0.039942, y_c + 0.100590, z_c, rx, ry, rz], a, v)
    movel(p[x_c + -0.039897, y_c + 0.100575, z_c, rx, ry, rz], a, v)
    movel(p[x_c + -0.039850, y_c + 0.100560, z_c, rx, ry, rz], a, v)
    movel(p[x_c + -0.039803, y_c + 0.100544, z_c, rx, ry, rz], a, v)
    movel(p[x_c + -0.039754, y_c + 0.100528, z_c, rx, ry, rz], a, v)
    movel(p[x_c + -0.039704, y_c + 0.100512, z_c, rx, ry, rz], a, v)
    movel(p[x_c + -0.039653, y_c + 0.100495, z_c, rx, ry, rz], a, v)
    movel(p[x_c + -0.039600, y_c + 0.100479, z_c, rx, ry, rz], a, v)
    movel(p[x_c + -0.039547, y_c + 0.100462, z_c, rx, ry, rz], a, v)
    movel(p[x_c + -0.039493, y_c + 0.100445, z_c, rx, ry, rz], a, v)
    movel(p[x_c + -0.039437, y_c + 0.100427, z_c, rx, ry, rz], a, v)
    movel(p[x_c + -0.039381, y_c + 0.100410, z_c, rx, ry, rz], a, v)
    movel(p[x_c + -0.039324, y_c + 0.100392, z_c, rx, ry, rz], a, v)
    movel(p[x_c + -0.039266, y_c + 0.100374, z_c, rx, ry, rz], a, v)
    movel(p[x_c + -0.039207, y_c + 0.100356, z_c, rx, ry, rz], a, v)
    movel(p[x_c + -0.039147, y_c + 0.100338, z_c, rx, ry, rz], a, v)
    movel(p[x_c + -0.039087, y_c + 0.100319, z_c, rx, ry, rz], a, v)
    movel(p[x_c + -0.039026, y_c + 0.100301, z_c, rx, ry, rz], a, v)
    movel(p[x_c + -0.038964, y_c + 0.100282, z_c, rx, ry, rz], a, v)
    movel(p[x_c + -0.038902, y_c + 0.100264, z_c, rx, ry, rz], a, v)
    movel(p[x_c + -0.038839, y_c + 0.100245, z_c, rx, ry, rz], a, v)
    movel(p[x_c + -0.038775, y_c + 0.100226, z_c, rx, ry, rz], a, v)
    movel(p[x_c + -0.038712, y_c + 0.100207, z_c, rx, ry, rz], a, v)
    movel(p[x_c + -0.038647, y_c + 0.100189, z_c, rx, ry, rz], a, v)
    movel(p[x_c + -0.038582, y_c + 0.100170, z_c, rx, ry, rz], a, v)
    movel(p[x_c + -0.038517, y_c + 0.100151, z_c, rx, ry, rz], a, v)
    movel(p[x_c + -0.038452, y_c + 0.100132, z_c, rx, ry, rz], a, v)
    movel(p[x_c + -0.038386, y_c + 0.100113, z_c, rx, ry, rz], a, v)
    movel(p[x_c + -0.038320, y_c + 0.100094, z_c, rx, ry, rz], a, v)
    movel(p[x_c + -0.038254, y_c + 0.100076, z_c, rx, ry, rz], a, v)
    movel(p[x_c + -0.038188, y_c + 0.100057, z_c, rx, ry, rz], a, v)
    movel(p[x_c + -0.038188, y_c + 0.100057, z_c, rx, ry, rz], a, v)
    movel(p[x_c + -0.038032, y_c + 0.100014, z_c, rx, ry, rz], a, v)
    movel(p[x_c + -0.037877, y_c + 0.099973, z_c, rx, ry, rz], a, v)
    movel(p[x_c + -0.037723, y_c + 0.099934, z_c, rx, ry, rz], a, v)
    movel(p[x_c + -0.037571, y_c + 0.099896, z_c, rx, ry, rz], a, v)
    movel(p[x_c + -0.037419, y_c + 0.099861, z_c, rx, ry, rz], a, v)
    movel(p[x_c + -0.037269, y_c + 0.099828, z_c, rx, ry, rz], a, v)
    movel(p[x_c + -0.037119, y_c + 0.099797, z_c, rx, ry, rz], a, v)
    movel(p[x_c + -0.036971, y_c + 0.099768, z_c, rx, ry, rz], a, v)
    movel(p[x_c + -0.036823, y_c + 0.099740, z_c, rx, ry, rz], a, v)
    movel(p[x_c + -0.036677, y_c + 0.099715, z_c, rx, ry, rz], a, v)
    movel(p[x_c + -0.036531, y_c + 0.099692, z_c, rx, ry, rz], a, v)
    movel(p[x_c + -0.036387, y_c + 0.099671, z_c, rx, ry, rz], a, v)
    movel(p[x_c + -0.036244, y_c + 0.099651, z_c, rx, ry, rz], a, v)
    movel(p[x_c + -0.036102, y_c + 0.099634, z_c, rx, ry, rz], a, v)
    movel(p[x_c + -0.035960, y_c + 0.099619, z_c, rx, ry, rz], a, v)
    movel(p[x_c + -0.035820, y_c + 0.099605, z_c, rx, ry, rz], a, v)
    movel(p[x_c + -0.035681, y_c + 0.099594, z_c, rx, ry, rz], a, v)
    movel(p[x_c + -0.035543, y_c + 0.099585, z_c, rx, ry, rz], a, v)
    movel(p[x_c + -0.035405, y_c + 0.099577, z_c, rx, ry, rz], a, v)
    movel(p[x_c + -0.035269, y_c + 0.099572, z_c, rx, ry, rz], a, v)
    movel(p[x_c + -0.035134, y_c + 0.099568, z_c, rx, ry, rz], a, v)
    movel(p[x_c + -0.035000, y_c + 0.099567, z_c, rx, ry, rz], a, v)
    movel(p[x_c + -0.034866, y_c + 0.099567, z_c, rx, ry, rz], a, v)
    movel(p[x_c + -0.034734, y_c + 0.099570, z_c, rx, ry, rz], a, v)
    movel(p[x_c + -0.034603, y_c + 0.099574, z_c, rx, ry, rz], a, v)
    movel(p[x_c + -0.034472, y_c + 0.099581, z_c, rx, ry, rz], a, v)
    movel(p[x_c + -0.034343, y_c + 0.099589, z_c, rx, ry, rz], a, v)
    movel(p[x_c + -0.034215, y_c + 0.099600, z_c, rx, ry, rz], a, v)
    movel(p[x_c + -0.034087, y_c + 0.099612, z_c, rx, ry, rz], a, v)
    movel(p[x_c + -0.033961, y_c + 0.099626, z_c, rx, ry, rz], a, v)
    movel(p[x_c + -0.033835, y_c + 0.099643, z_c, rx, ry, rz], a, v)
    movel(p[x_c + -0.033711, y_c + 0.099661, z_c, rx, ry, rz], a, v)
    movel(p[x_c + -0.033587, y_c + 0.099681, z_c, rx, ry, rz], a, v)
    movel(p[x_c + -0.033464, y_c + 0.099704, z_c, rx, ry, rz], a, v)
    movel(p[x_c + -0.033343, y_c + 0.099728, z_c, rx, ry, rz], a, v)
    movel(p[x_c + -0.033222, y_c + 0.099754, z_c, rx, ry, rz], a, v)
    movel(p[x_c + -0.033102, y_c + 0.099783, z_c, rx, ry, rz], a, v)
    movel(p[x_c + -0.032983, y_c + 0.099813, z_c, rx, ry, rz], a, v)
    movel(p[x_c + -0.032865, y_c + 0.099845, z_c, rx, ry, rz], a, v)
    movel(p[x_c + -0.032748, y_c + 0.099879, z_c, rx, ry, rz], a, v)
    movel(p[x_c + -0.032632, y_c + 0.099916, z_c, rx, ry, rz], a, v)
    movel(p[x_c + -0.032517, y_c + 0.099954, z_c, rx, ry, rz], a, v)
    movel(p[x_c + -0.032402, y_c + 0.099994, z_c, rx, ry, rz], a, v)
    movel(p[x_c + -0.032289, y_c + 0.100036, z_c, rx, ry, rz], a, v)
    movel(p[x_c + -0.032176, y_c + 0.100080, z_c, rx, ry, rz], a, v)
    movel(p[x_c + -0.032065, y_c + 0.100127, z_c, rx, ry, rz], a, v)
    movel(p[x_c + -0.031954, y_c + 0.100175, z_c, rx, ry, rz], a, v)
    movel(p[x_c + -0.031844, y_c + 0.100225, z_c, rx, ry, rz], a, v)
    movel(p[x_c + -0.031735, y_c + 0.100277, z_c, rx, ry, rz], a, v)
    movel(p[x_c + -0.031735, y_c + 0.100277, z_c, rx, ry, rz], a, v)
    movel(p[x_c + -0.031735, y_c + 0.100277, z_c, rx, ry, rz], a, v)
    movel(p[x_c + -0.031735, y_c + 0.100277, z_c, rx, ry, rz], a, v)
    movel(p[x_c + -0.031735, y_c + 0.100277, z_c, rx, ry, rz], a, v)
    movel(p[x_c + -0.031735, y_c + 0.100277, z_c, rx, ry, rz], a, v)
    movel(p[x_c + -0.031735, y_c + 0.100277, z_c, rx, ry, rz], a, v)
    movel(p[x_c + -0.031735, y_c + 0.100277, z_c, rx, ry, rz], a, v)
    movel(p[x_c + -0.031735, y_c + 0.100277, z_c, rx, ry, rz], a, v)
    movel(p[x_c + -0.031735, y_c + 0.100277, z_c, rx, ry, rz], a, v)
    movel(p[x_c + -0.031735, y_c + 0.100277, z_c, rx, ry, rz], a, v)
    movel(p[x_c + -0.036942, y_c + 0.100761, z_c, rx, ry, rz], a, v)
    movel(p[x_c + -0.036942, y_c + 0.100761, z_c, rx, ry, rz], a, v)
    movel(p[x_c + -0.036942, y_c + 0.100761, z_c, rx, ry, rz], a, v)
    movel(p[x_c + -0.036942, y_c + 0.100761, z_c, rx, ry, rz], a, v)
    movel(p[x_c + -0.036942, y_c + 0.100761, z_c, rx, ry, rz], a, v)
    movel(p[x_c + -0.036942, y_c + 0.100761, z_c, rx, ry, rz], a, v)
    movel(p[x_c + -0.036942, y_c + 0.100761, z_c, rx, ry, rz], a, v)
    movel(p[x_c + -0.036942, y_c + 0.100761, z_c, rx, ry, rz], a, v)
    movel(p[x_c + -0.036942, y_c + 0.100761, z_c, rx, ry, rz], a, v)
    movel(p[x_c + -0.036942, y_c + 0.100761, z_c, rx, ry, rz], a, v)
    movel(p[x_c + -0.036942, y_c + 0.100761, z_c, rx, ry, rz], a, v)
    movel(p[x_c + -0.036973, y_c + 0.100772, z_c, rx, ry, rz], a, v)
    movel(p[x_c + -0.037005, y_c + 0.100784, z_c, rx, ry, rz], a, v)
    movel(p[x_c + -0.037036, y_c + 0.100795, z_c, rx, ry, rz], a, v)
    movel(p[x_c + -0.037067, y_c + 0.100807, z_c, rx, ry, rz], a, v)
    movel(p[x_c + -0.037098, y_c + 0.100819, z_c, rx, ry, rz], a, v)
    movel(p[x_c + -0.037128, y_c + 0.100831, z_c, rx, ry, rz], a, v)
    movel(p[x_c + -0.037158, y_c + 0.100842, z_c, rx, ry, rz], a, v)
    movel(p[x_c + -0.037188, y_c + 0.100854, z_c, rx, ry, rz], a, v)
    movel(p[x_c + -0.037217, y_c + 0.100866, z_c, rx, ry, rz], a, v)
    movel(p[x_c + -0.037246, y_c + 0.100878, z_c, rx, ry, rz], a, v)
    movel(p[x_c + -0.037275, y_c + 0.100890, z_c, rx, ry, rz], a, v)
    movel(p[x_c + -0.037303, y_c + 0.100902, z_c, rx, ry, rz], a, v)
    movel(p[x_c + -0.037331, y_c + 0.100914, z_c, rx, ry, rz], a, v)
    movel(p[x_c + -0.037358, y_c + 0.100925, z_c, rx, ry, rz], a, v)
    movel(p[x_c + -0.037384, y_c + 0.100937, z_c, rx, ry, rz], a, v)
    movel(p[x_c + -0.037411, y_c + 0.100949, z_c, rx, ry, rz], a, v)
    movel(p[x_c + -0.037436, y_c + 0.100961, z_c, rx, ry, rz], a, v)
    movel(p[x_c + -0.037462, y_c + 0.100973, z_c, rx, ry, rz], a, v)
    movel(p[x_c + -0.037486, y_c + 0.100984, z_c, rx, ry, rz], a, v)
    movel(p[x_c + -0.037510, y_c + 0.100996, z_c, rx, ry, rz], a, v)
    movel(p[x_c + -0.037534, y_c + 0.101007, z_c, rx, ry, rz], a, v)
    movel(p[x_c + -0.037557, y_c + 0.101019, z_c, rx, ry, rz], a, v)
    movel(p[x_c + -0.037579, y_c + 0.101030, z_c, rx, ry, rz], a, v)
    movel(p[x_c + -0.037601, y_c + 0.101042, z_c, rx, ry, rz], a, v)
    movel(p[x_c + -0.037622, y_c + 0.101053, z_c, rx, ry, rz], a, v)
    movel(p[x_c + -0.037642, y_c + 0.101064, z_c, rx, ry, rz], a, v)
    movel(p[x_c + -0.037662, y_c + 0.101075, z_c, rx, ry, rz], a, v)
    movel(p[x_c + -0.037681, y_c + 0.101085, z_c, rx, ry, rz], a, v)
    movel(p[x_c + -0.037699, y_c + 0.101096, z_c, rx, ry, rz], a, v)
    movel(p[x_c + -0.037717, y_c + 0.101106, z_c, rx, ry, rz], a, v)
    movel(p[x_c + -0.037734, y_c + 0.101117, z_c, rx, ry, rz], a, v)
    movel(p[x_c + -0.037750, y_c + 0.101127, z_c, rx, ry, rz], a, v)
    movel(p[x_c + -0.037765, y_c + 0.101137, z_c, rx, ry, rz], a, v)
    movel(p[x_c + -0.037780, y_c + 0.101146, z_c, rx, ry, rz], a, v)
    movel(p[x_c + -0.037793, y_c + 0.101156, z_c, rx, ry, rz], a, v)
    movel(p[x_c + -0.037806, y_c + 0.101165, z_c, rx, ry, rz], a, v)
    movel(p[x_c + -0.037818, y_c + 0.101174, z_c, rx, ry, rz], a, v)
    movel(p[x_c + -0.037829, y_c + 0.101183, z_c, rx, ry, rz], a, v)
    movel(p[x_c + -0.037840, y_c + 0.101192, z_c, rx, ry, rz], a, v)
    movel(p[x_c + -0.037849, y_c + 0.101200, z_c, rx, ry, rz], a, v)
    movel(p[x_c + -0.037857, y_c + 0.101208, z_c, rx, ry, rz], a, v)
    movel(p[x_c + -0.037865, y_c + 0.101216, z_c, rx, ry, rz], a, v)
    movel(p[x_c + -0.037872, y_c + 0.101224, z_c, rx, ry, rz], a, v)
    movel(p[x_c + -0.037877, y_c + 0.101231, z_c, rx, ry, rz], a, v)
    movel(p[x_c + -0.037882, y_c + 0.101238, z_c, rx, ry, rz], a, v)
    movel(p[x_c + -0.037885, y_c + 0.101245, z_c, rx, ry, rz], a, v)
    movel(p[x_c + -0.037888, y_c + 0.101251, z_c, rx, ry, rz], a, v)
    movel(p[x_c + -0.037890, y_c + 0.101257, z_c, rx, ry, rz], a, v)
    movel(p[x_c + -0.037890, y_c + 0.101263, z_c, rx, ry, rz], a, v)
    movel(p[x_c + -0.037890, y_c + 0.101263, z_c, rx, ry, rz], a, v)
    movel(p[x_c + -0.037887, y_c + 0.101278, z_c, rx, ry, rz], a, v)
    movel(p[x_c + -0.037878, y_c + 0.101297, z_c, rx, ry, rz], a, v)
    movel(p[x_c + -0.037862, y_c + 0.101320, z_c, rx, ry, rz], a, v)
    movel(p[x_c + -0.037841, y_c + 0.101348, z_c, rx, ry, rz], a, v)
    movel(p[x_c + -0.037814, y_c + 0.101380, z_c, rx, ry, rz], a, v)
    movel(p[x_c + -0.037782, y_c + 0.101416, z_c, rx, ry, rz], a, v)
    movel(p[x_c + -0.037744, y_c + 0.101455, z_c, rx, ry, rz], a, v)
    movel(p[x_c + -0.037702, y_c + 0.101498, z_c, rx, ry, rz], a, v)
    movel(p[x_c + -0.037656, y_c + 0.101544, z_c, rx, ry, rz], a, v)
    movel(p[x_c + -0.037604, y_c + 0.101593, z_c, rx, ry, rz], a, v)
    movel(p[x_c + -0.037549, y_c + 0.101646, z_c, rx, ry, rz], a, v)
    movel(p[x_c + -0.037490, y_c + 0.101700, z_c, rx, ry, rz], a, v)
    movel(p[x_c + -0.037426, y_c + 0.101758, z_c, rx, ry, rz], a, v)
    movel(p[x_c + -0.037360, y_c + 0.101817, z_c, rx, ry, rz], a, v)
    movel(p[x_c + -0.037290, y_c + 0.101879, z_c, rx, ry, rz], a, v)
    movel(p[x_c + -0.037217, y_c + 0.101943, z_c, rx, ry, rz], a, v)
    movel(p[x_c + -0.037141, y_c + 0.102009, z_c, rx, ry, rz], a, v)
    movel(p[x_c + -0.037063, y_c + 0.102076, z_c, rx, ry, rz], a, v)
    movel(p[x_c + -0.036982, y_c + 0.102144, z_c, rx, ry, rz], a, v)
    movel(p[x_c + -0.036899, y_c + 0.102214, z_c, rx, ry, rz], a, v)
    movel(p[x_c + -0.036815, y_c + 0.102285, z_c, rx, ry, rz], a, v)
    movel(p[x_c + -0.036728, y_c + 0.102357, z_c, rx, ry, rz], a, v)
    movel(p[x_c + -0.036641, y_c + 0.102429, z_c, rx, ry, rz], a, v)
    movel(p[x_c + -0.036552, y_c + 0.102502, z_c, rx, ry, rz], a, v)
    movel(p[x_c + -0.036462, y_c + 0.102575, z_c, rx, ry, rz], a, v)
    movel(p[x_c + -0.036371, y_c + 0.102649, z_c, rx, ry, rz], a, v)
    movel(p[x_c + -0.036280, y_c + 0.102722, z_c, rx, ry, rz], a, v)
    movel(p[x_c + -0.036188, y_c + 0.102795, z_c, rx, ry, rz], a, v)
    movel(p[x_c + -0.036096, y_c + 0.102867, z_c, rx, ry, rz], a, v)
    movel(p[x_c + -0.036005, y_c + 0.102939, z_c, rx, ry, rz], a, v)
    movel(p[x_c + -0.035914, y_c + 0.103010, z_c, rx, ry, rz], a, v)
    movel(p[x_c + -0.035823, y_c + 0.103080, z_c, rx, ry, rz], a, v)
    movel(p[x_c + -0.035734, y_c + 0.103149, z_c, rx, ry, rz], a, v)
    movel(p[x_c + -0.035645, y_c + 0.103216, z_c, rx, ry, rz], a, v)
    movel(p[x_c + -0.035558, y_c + 0.103282, z_c, rx, ry, rz], a, v)
    movel(p[x_c + -0.035472, y_c + 0.103346, z_c, rx, ry, rz], a, v)
    movel(p[x_c + -0.035389, y_c + 0.103409, z_c, rx, ry, rz], a, v)
    movel(p[x_c + -0.035307, y_c + 0.103469, z_c, rx, ry, rz], a, v)
    movel(p[x_c + -0.035227, y_c + 0.103526, z_c, rx, ry, rz], a, v)
    movel(p[x_c + -0.035150, y_c + 0.103582, z_c, rx, ry, rz], a, v)
    movel(p[x_c + -0.035075, y_c + 0.103634, z_c, rx, ry, rz], a, v)
    movel(p[x_c + -0.035004, y_c + 0.103684, z_c, rx, ry, rz], a, v)
    movel(p[x_c + -0.034935, y_c + 0.103730, z_c, rx, ry, rz], a, v)
    movel(p[x_c + -0.034870, y_c + 0.103774, z_c, rx, ry, rz], a, v)
    movel(p[x_c + -0.034809, y_c + 0.103814, z_c, rx, ry, rz], a, v)
    movel(p[x_c + -0.034751, y_c + 0.103850, z_c, rx, ry, rz], a, v)
    movel(p[x_c + -0.034698, y_c + 0.103882, z_c, rx, ry, rz], a, v)
    movel(p[x_c + -0.034648, y_c + 0.103911, z_c, rx, ry, rz], a, v)
    movel(p[x_c + -0.034603, y_c + 0.103935, z_c, rx, ry, rz], a, v)
    movel(p[x_c + -0.034603, y_c + 0.103935, z_c, rx, ry, rz], a, v)
    movel(p[x_c + -0.034549, y_c + 0.103963, z_c, rx, ry, rz], a, v)
    movel(p[x_c + -0.034492, y_c + 0.103990, z_c, rx, ry, rz], a, v)
    movel(p[x_c + -0.034433, y_c + 0.104016, z_c, rx, ry, rz], a, v)
    movel(p[x_c + -0.034371, y_c + 0.104042, z_c, rx, ry, rz], a, v)
    movel(p[x_c + -0.034306, y_c + 0.104068, z_c, rx, ry, rz], a, v)
    movel(p[x_c + -0.034240, y_c + 0.104093, z_c, rx, ry, rz], a, v)
    movel(p[x_c + -0.034171, y_c + 0.104117, z_c, rx, ry, rz], a, v)
    movel(p[x_c + -0.034100, y_c + 0.104141, z_c, rx, ry, rz], a, v)
    movel(p[x_c + -0.034028, y_c + 0.104165, z_c, rx, ry, rz], a, v)
    movel(p[x_c + -0.033953, y_c + 0.104188, z_c, rx, ry, rz], a, v)
    movel(p[x_c + -0.033876, y_c + 0.104210, z_c, rx, ry, rz], a, v)
    movel(p[x_c + -0.033798, y_c + 0.104231, z_c, rx, ry, rz], a, v)
    movel(p[x_c + -0.033718, y_c + 0.104253, z_c, rx, ry, rz], a, v)
    movel(p[x_c + -0.033637, y_c + 0.104273, z_c, rx, ry, rz], a, v)
    movel(p[x_c + -0.033554, y_c + 0.104293, z_c, rx, ry, rz], a, v)
    movel(p[x_c + -0.033469, y_c + 0.104312, z_c, rx, ry, rz], a, v)
    movel(p[x_c + -0.033384, y_c + 0.104330, z_c, rx, ry, rz], a, v)
    movel(p[x_c + -0.033297, y_c + 0.104348, z_c, rx, ry, rz], a, v)
    movel(p[x_c + -0.033209, y_c + 0.104366, z_c, rx, ry, rz], a, v)
    movel(p[x_c + -0.033120, y_c + 0.104382, z_c, rx, ry, rz], a, v)
    movel(p[x_c + -0.033030, y_c + 0.104398, z_c, rx, ry, rz], a, v)
    movel(p[x_c + -0.032939, y_c + 0.104413, z_c, rx, ry, rz], a, v)
    movel(p[x_c + -0.032847, y_c + 0.104427, z_c, rx, ry, rz], a, v)
    movel(p[x_c + -0.032755, y_c + 0.104441, z_c, rx, ry, rz], a, v)
    movel(p[x_c + -0.032662, y_c + 0.104454, z_c, rx, ry, rz], a, v)
    movel(p[x_c + -0.032568, y_c + 0.104466, z_c, rx, ry, rz], a, v)
    movel(p[x_c + -0.032474, y_c + 0.104477, z_c, rx, ry, rz], a, v)
    movel(p[x_c + -0.032380, y_c + 0.104488, z_c, rx, ry, rz], a, v)
    movel(p[x_c + -0.032285, y_c + 0.104498, z_c, rx, ry, rz], a, v)
    movel(p[x_c + -0.032190, y_c + 0.104507, z_c, rx, ry, rz], a, v)
    movel(p[x_c + -0.032095, y_c + 0.104515, z_c, rx, ry, rz], a, v)
    movel(p[x_c + -0.032000, y_c + 0.104522, z_c, rx, ry, rz], a, v)
    movel(p[x_c + -0.031905, y_c + 0.104528, z_c, rx, ry, rz], a, v)
    movel(p[x_c + -0.031811, y_c + 0.104534, z_c, rx, ry, rz], a, v)
    movel(p[x_c + -0.031716, y_c + 0.104539, z_c, rx, ry, rz], a, v)
    movel(p[x_c + -0.031622, y_c + 0.104543, z_c, rx, ry, rz], a, v)
    movel(p[x_c + -0.031528, y_c + 0.104546, z_c, rx, ry, rz], a, v)
    movel(p[x_c + -0.031435, y_c + 0.104548, z_c, rx, ry, rz], a, v)
    movel(p[x_c + -0.031342, y_c + 0.104549, z_c, rx, ry, rz], a, v)
    movel(p[x_c + -0.031250, y_c + 0.104549, z_c, rx, ry, rz], a, v)
    movel(p[x_c + -0.031159, y_c + 0.104549, z_c, rx, ry, rz], a, v)
    movel(p[x_c + -0.031068, y_c + 0.104547, z_c, rx, ry, rz], a, v)
    movel(p[x_c + -0.030979, y_c + 0.104544, z_c, rx, ry, rz], a, v)
    movel(p[x_c + -0.030890, y_c + 0.104541, z_c, rx, ry, rz], a, v)
    movel(p[x_c + -0.030803, y_c + 0.104536, z_c, rx, ry, rz], a, v)
    movel(p[x_c + -0.030717, y_c + 0.104531, z_c, rx, ry, rz], a, v)
    movel(p[x_c + -0.030632, y_c + 0.104524, z_c, rx, ry, rz], a, v)
    movel(p[x_c + -0.030548, y_c + 0.104516, z_c, rx, ry, rz], a, v)
    movel(p[x_c + -0.030466, y_c + 0.104508, z_c, rx, ry, rz], a, v)
    movel(p[x_c + -0.030466, y_c + 0.104508, z_c, rx, ry, rz], a, v)
    movel(p[x_c + -0.029180, y_c + 0.104364, z_c, rx, ry, rz], a, v)
    movel(p[x_c + -0.029180, y_c + 0.104364, z_c, rx, ry, rz], a, v)
    movel(p[x_c + -0.029685, y_c + 0.103464, z_c, rx, ry, rz], a, v)
    movel(p[x_c + -0.029685, y_c + 0.103464, z_c, rx, ry, rz], a, v)
    movel(p[x_c + -0.029773, y_c + 0.103313, z_c, rx, ry, rz], a, v)
    movel(p[x_c + -0.029865, y_c + 0.103165, z_c, rx, ry, rz], a, v)
    movel(p[x_c + -0.029961, y_c + 0.103021, z_c, rx, ry, rz], a, v)
    movel(p[x_c + -0.030061, y_c + 0.102880, z_c, rx, ry, rz], a, v)
    movel(p[x_c + -0.030165, y_c + 0.102743, z_c, rx, ry, rz], a, v)
    movel(p[x_c + -0.030273, y_c + 0.102609, z_c, rx, ry, rz], a, v)
    movel(p[x_c + -0.030384, y_c + 0.102478, z_c, rx, ry, rz], a, v)
    movel(p[x_c + -0.030499, y_c + 0.102352, z_c, rx, ry, rz], a, v)
    movel(p[x_c + -0.030618, y_c + 0.102228, z_c, rx, ry, rz], a, v)
    movel(p[x_c + -0.030740, y_c + 0.102109, z_c, rx, ry, rz], a, v)
    movel(p[x_c + -0.030865, y_c + 0.101993, z_c, rx, ry, rz], a, v)
    movel(p[x_c + -0.030994, y_c + 0.101881, z_c, rx, ry, rz], a, v)
    movel(p[x_c + -0.031125, y_c + 0.101773, z_c, rx, ry, rz], a, v)
    movel(p[x_c + -0.031259, y_c + 0.101669, z_c, rx, ry, rz], a, v)
    movel(p[x_c + -0.031396, y_c + 0.101568, z_c, rx, ry, rz], a, v)
    movel(p[x_c + -0.031536, y_c + 0.101472, z_c, rx, ry, rz], a, v)
    movel(p[x_c + -0.031679, y_c + 0.101379, z_c, rx, ry, rz], a, v)
    movel(p[x_c + -0.031823, y_c + 0.101291, z_c, rx, ry, rz], a, v)
    movel(p[x_c + -0.031971, y_c + 0.101206, z_c, rx, ry, rz], a, v)
    movel(p[x_c + -0.032120, y_c + 0.101126, z_c, rx, ry, rz], a, v)
    movel(p[x_c + -0.032272, y_c + 0.101050, z_c, rx, ry, rz], a, v)
    movel(p[x_c + -0.032426, y_c + 0.100978, z_c, rx, ry, rz], a, v)
    movel(p[x_c + -0.032581, y_c + 0.100910, z_c, rx, ry, rz], a, v)
    movel(p[x_c + -0.032739, y_c + 0.100846, z_c, rx, ry, rz], a, v)
    movel(p[x_c + -0.032898, y_c + 0.100787, z_c, rx, ry, rz], a, v)
    movel(p[x_c + -0.033059, y_c + 0.100732, z_c, rx, ry, rz], a, v)
    movel(p[x_c + -0.033221, y_c + 0.100682, z_c, rx, ry, rz], a, v)
    movel(p[x_c + -0.033384, y_c + 0.100635, z_c, rx, ry, rz], a, v)
    movel(p[x_c + -0.033549, y_c + 0.100594, z_c, rx, ry, rz], a, v)
    movel(p[x_c + -0.033715, y_c + 0.100557, z_c, rx, ry, rz], a, v)
    movel(p[x_c + -0.033882, y_c + 0.100524, z_c, rx, ry, rz], a, v)
    movel(p[x_c + -0.034050, y_c + 0.100496, z_c, rx, ry, rz], a, v)
    movel(p[x_c + -0.034219, y_c + 0.100473, z_c, rx, ry, rz], a, v)
    movel(p[x_c + -0.034389, y_c + 0.100454, z_c, rx, ry, rz], a, v)
    movel(p[x_c + -0.034559, y_c + 0.100440, z_c, rx, ry, rz], a, v)
    movel(p[x_c + -0.034729, y_c + 0.100431, z_c, rx, ry, rz], a, v)
    movel(p[x_c + -0.034900, y_c + 0.100426, z_c, rx, ry, rz], a, v)
    movel(p[x_c + -0.035072, y_c + 0.100426, z_c, rx, ry, rz], a, v)
    movel(p[x_c + -0.035243, y_c + 0.100432, z_c, rx, ry, rz], a, v)
    movel(p[x_c + -0.035414, y_c + 0.100442, z_c, rx, ry, rz], a, v)
    movel(p[x_c + -0.035586, y_c + 0.100457, z_c, rx, ry, rz], a, v)
    movel(p[x_c + -0.035757, y_c + 0.100477, z_c, rx, ry, rz], a, v)
    movel(p[x_c + -0.035928, y_c + 0.100502, z_c, rx, ry, rz], a, v)
    movel(p[x_c + -0.036099, y_c + 0.100532, z_c, rx, ry, rz], a, v)
    movel(p[x_c + -0.036269, y_c + 0.100568, z_c, rx, ry, rz], a, v)
    movel(p[x_c + -0.036438, y_c + 0.100608, z_c, rx, ry, rz], a, v)
    movel(p[x_c + -0.036607, y_c + 0.100654, z_c, rx, ry, rz], a, v)
    movel(p[x_c + -0.036775, y_c + 0.100705, z_c, rx, ry, rz], a, v)
    movel(p[x_c + -0.036942, y_c + 0.100761, z_c, rx, ry, rz], a, v)
    movel(p[x_c + -0.036942, y_c + 0.100761, z_c, rx, ry, rz], a, v)
    movel(p[x_c + -0.036942, y_c + 0.100761, z_c, rx, ry, rz], a, v)
    movel(p[x_c + -0.036942, y_c + 0.100761, z_c, rx, ry, rz], a, v)
    movel(p[x_c + -0.036942, y_c + 0.100761, z_c, rx, ry, rz], a, v)
    movel(p[x_c + -0.036942, y_c + 0.100761, z_c, rx, ry, rz], a, v)
    movel(p[x_c + -0.036942, y_c + 0.100761, z_c, rx, ry, rz], a, v)
    movel(p[x_c + -0.036942, y_c + 0.100761, z_c, rx, ry, rz], a, v)
    movel(p[x_c + -0.036942, y_c + 0.100761, z_c, rx, ry, rz], a, v)
    movel(p[x_c + -0.036942, y_c + 0.100761, z_c, rx, ry, rz], a, v)
    movel(p[x_c + -0.036942, y_c + 0.100761, z_c, rx, ry, rz], a, v)

    # Lift pen at end
    movel(p[x_c, y_c, z_c + z_lift, rx, ry, rz], a, v)
end

draw_image()
